  PROC DrawPart276()
    MoveL Offs(pOrigin,208.02,110.33,6.00),vTravel,z5,tPen\WObj:=wPaper;
    MoveL Offs(pOrigin,208.02,110.33,0.00),v60,z0,tPen\WObj:=wPaper;
    MoveL Offs(pOrigin,210.27,108.07,0.00),v40,fine,tPen\WObj:=wPaper;
    MoveL Offs(pOrigin,210.27,108.07,6.00),v60,z5,tPen\WObj:=wPaper;
    MoveL Offs(pOrigin,213.02,105.82,6.00),vTravel,z5,tPen\WObj:=wPaper;
    MoveL Offs(pOrigin,213.02,105.82,0.00),v60,z0,tPen\WObj:=wPaper;
    MoveL Offs(pOrigin,214.30,105.82,0.00),v40,fine,tPen\WObj:=wPaper;
    MoveL Offs(pOrigin,214.30,105.82,6.00),v60,z5,tPen\WObj:=wPaper;
    MoveL Offs(pOrigin,214.72,103.70,6.00),vTravel,z5,tPen\WObj:=wPaper;
    MoveL Offs(pOrigin,214.72,103.70,0.00),v60,z0,tPen\WObj:=wPaper;
    MoveL Offs(pOrigin,213.45,103.70,0.00),v40,z0,tPen\WObj:=wPaper;
    MoveL Offs(pOrigin,213.88,102.65,0.00),v40,z0,tPen\WObj:=wPaper;
    MoveL Offs(pOrigin,214.94,102.65,0.00),v40,fine,tPen\WObj:=wPaper;
    MoveL Offs(pOrigin,214.94,102.65,6.00),v60,z5,tPen\WObj:=wPaper;
    MoveL Offs(pOrigin,215.36,100.54,6.00),vTravel,z5,tPen\WObj:=wPaper;
    MoveL Offs(pOrigin,215.36,100.54,0.00),v60,z0,tPen\WObj:=wPaper;
    MoveL Offs(pOrigin,214.30,100.54,0.00),v40,z0,tPen\WObj:=wPaper;
    MoveL Offs(pOrigin,214.51,99.48,0.00),v40,z0,tPen\WObj:=wPaper;
    MoveL Offs(pOrigin,215.58,99.48,0.00),v40,z0,tPen\WObj:=wPaper;
    MoveL Offs(pOrigin,215.79,98.42,0.00),v40,z0,tPen\WObj:=wPaper;
    MoveL Offs(pOrigin,214.72,98.42,0.00),v40,fine,tPen\WObj:=wPaper;
    MoveL Offs(pOrigin,214.72,98.42,6.00),v60,z5,tPen\WObj:=wPaper;
    MoveL Offs(pOrigin,206.17,76.33,6.00),vTravel,z5,tPen\WObj:=wPaper;
    MoveL Offs(pOrigin,206.17,76.33,0.00),v60,z0,tPen\WObj:=wPaper;
    MoveL Offs(pOrigin,211.13,71.37,0.00),v40,z0,tPen\WObj:=wPaper;
    MoveL Offs(pOrigin,211.85,71.76,0.00),v40,z0,tPen\WObj:=wPaper;
    MoveL Offs(pOrigin,213.50,73.41,0.00),v40,fine,tPen\WObj:=wPaper;
    MoveL Offs(pOrigin,213.50,73.41,6.00),v60,z5,tPen\WObj:=wPaper;
    MoveL Offs(pOrigin,205.72,76.08,6.00),vTravel,z5,tPen\WObj:=wPaper;
    MoveL Offs(pOrigin,205.72,76.08,0.00),v60,z0,tPen\WObj:=wPaper;
    MoveL Offs(pOrigin,203.91,74.28,0.00),v40,fine,tPen\WObj:=wPaper;
    MoveL Offs(pOrigin,203.91,74.28,6.00),v60,z5,tPen\WObj:=wPaper;
    MoveL Offs(pOrigin,199.85,71.72,6.00),vTravel,z5,tPen\WObj:=wPaper;
    MoveL Offs(pOrigin,199.85,71.72,0.00),v60,z0,tPen\WObj:=wPaper;
    MoveL Offs(pOrigin,200.27,71.51,0.00),v40,z0,tPen\WObj:=wPaper;
    MoveL Offs(pOrigin,199.85,71.72,0.00),v40,fine,tPen\WObj:=wPaper;
    MoveL Offs(pOrigin,199.85,71.72,6.00),v60,z5,tPen\WObj:=wPaper;
    MoveL Offs(pOrigin,196.43,72.15,6.00),vTravel,z5,tPen\WObj:=wPaper;
    MoveL Offs(pOrigin,196.43,72.15,0.00),v60,z0,tPen\WObj:=wPaper;
    MoveL Offs(pOrigin,196.43,75.76,0.00),v40,fine,tPen\WObj:=wPaper;
    MoveL Offs(pOrigin,196.43,75.76,6.00),v60,z5,tPen\WObj:=wPaper;
    MoveL Offs(pOrigin,194.75,76.40,6.00),vTravel,z5,tPen\WObj:=wPaper;
    MoveL Offs(pOrigin,194.75,76.40,0.00),v60,z0,tPen\WObj:=wPaper;
    MoveL Offs(pOrigin,194.32,76.82,0.00),v40,z0,tPen\WObj:=wPaper;
    MoveL Offs(pOrigin,194.75,76.40,0.00),v40,z0,tPen\WObj:=wPaper;
    MoveL Offs(pOrigin,194.32,76.19,0.00),v40,z0,tPen\WObj:=wPaper;
    MoveL Offs(pOrigin,194.32,73.64,0.00),v40,z0,tPen\WObj:=wPaper;
    MoveL Offs(pOrigin,193.26,73.85,0.00),v40,z0,tPen\WObj:=wPaper;
    MoveL Offs(pOrigin,193.26,74.91,0.00),v40,fine,tPen\WObj:=wPaper;
    MoveL Offs(pOrigin,193.26,74.91,6.00),v60,z5,tPen\WObj:=wPaper;
    MoveL Offs(pOrigin,194.11,77.04,6.00),vTravel,z5,tPen\WObj:=wPaper;
    MoveL Offs(pOrigin,194.11,77.04,0.00),v60,z0,tPen\WObj:=wPaper;
    MoveL Offs(pOrigin,193.69,77.46,0.00),v40,z0,tPen\WObj:=wPaper;
    MoveL Offs(pOrigin,194.11,77.04,0.00),v40,z0,tPen\WObj:=wPaper;
    MoveL Offs(pOrigin,194.79,77.10,0.00),v40,z0,tPen\WObj:=wPaper;
    MoveL Offs(pOrigin,191.33,73.64,0.00),v40,fine,tPen\WObj:=wPaper;
    MoveL Offs(pOrigin,191.33,73.64,6.00),v60,z5,tPen\WObj:=wPaper;
    MoveL Offs(pOrigin,189.24,74.54,6.00),vTravel,z5,tPen\WObj:=wPaper;
    MoveL Offs(pOrigin,189.24,74.54,0.00),v60,z0,tPen\WObj:=wPaper;
    MoveL Offs(pOrigin,193.14,78.44,0.00),v40,z0,tPen\WObj:=wPaper;
    MoveL Offs(pOrigin,193.05,77.89,0.00),v40,z0,tPen\WObj:=wPaper;
    MoveL Offs(pOrigin,191.77,79.16,0.00),v40,z0,tPen\WObj:=wPaper;
    MoveL Offs(pOrigin,193.05,77.89,0.00),v40,z0,tPen\WObj:=wPaper;
    MoveL Offs(pOrigin,192.20,78.36,0.00),v40,z0,tPen\WObj:=wPaper;
    MoveL Offs(pOrigin,188.80,78.36,0.00),v40,fine,tPen\WObj:=wPaper;
    MoveL Offs(pOrigin,188.80,78.36,6.00),v60,z5,tPen\WObj:=wPaper;
    MoveL Offs(pOrigin,190.09,78.52,6.00),vTravel,z5,tPen\WObj:=wPaper;
    MoveL Offs(pOrigin,190.09,78.52,0.00),v60,z0,tPen\WObj:=wPaper;
    MoveL Offs(pOrigin,190.09,79.59,0.00),v40,z0,tPen\WObj:=wPaper;
    MoveL Offs(pOrigin,190.08,80.47,0.00),v40,z0,tPen\WObj:=wPaper;
    MoveL Offs(pOrigin,187.31,80.47,0.00),v40,z0,tPen\WObj:=wPaper;
    MoveL Offs(pOrigin,186.26,80.52,0.00),v40,z0,tPen\WObj:=wPaper;
    MoveL Offs(pOrigin,188.81,83.07,0.00),v40,z0,tPen\WObj:=wPaper;
    MoveL Offs(pOrigin,188.80,82.78,0.00),v40,z0,tPen\WObj:=wPaper;
    MoveL Offs(pOrigin,187.52,84.05,0.00),v40,z0,tPen\WObj:=wPaper;
    MoveL Offs(pOrigin,188.80,82.78,0.00),v40,z0,tPen\WObj:=wPaper;
    MoveL Offs(pOrigin,188.59,82.58,0.00),v40,z0,tPen\WObj:=wPaper;
    MoveL Offs(pOrigin,186.25,82.58,0.00),v40,fine,tPen\WObj:=wPaper;
    MoveL Offs(pOrigin,186.25,82.58,6.00),v60,z5,tPen\WObj:=wPaper;
    MoveL Offs(pOrigin,185.51,81.27,6.00),vTravel,z5,tPen\WObj:=wPaper;
    MoveL Offs(pOrigin,185.51,81.27,0.00),v60,z0,tPen\WObj:=wPaper;
    MoveL Offs(pOrigin,188.22,83.97,0.00),v40,fine,tPen\WObj:=wPaper;
    MoveL Offs(pOrigin,188.22,83.97,6.00),v60,z5,tPen\WObj:=wPaper;
    MoveL Offs(pOrigin,190.31,81.58,6.00),vTravel,z5,tPen\WObj:=wPaper;
    MoveL Offs(pOrigin,190.31,81.58,0.00),v60,z0,tPen\WObj:=wPaper;
    MoveL Offs(pOrigin,187.60,78.87,0.00),v40,fine,tPen\WObj:=wPaper;
    MoveL Offs(pOrigin,187.60,78.87,6.00),v60,z5,tPen\WObj:=wPaper;
    MoveL Offs(pOrigin,183.56,80.81,6.00),vTravel,z5,tPen\WObj:=wPaper;
    MoveL Offs(pOrigin,183.56,80.81,0.00),v60,z0,tPen\WObj:=wPaper;
    MoveL Offs(pOrigin,179.35,76.60,0.00),v40,z0,tPen\WObj:=wPaper;
    MoveL Offs(pOrigin,179.51,76.11,0.00),v40,z0,tPen\WObj:=wPaper;
    MoveL Offs(pOrigin,177.11,78.52,0.00),v40,z0,tPen\WObj:=wPaper;
    MoveL Offs(pOrigin,176.21,77.92,0.00),v40,z0,tPen\WObj:=wPaper;
    MoveL Offs(pOrigin,178.46,75.67,0.00),v40,fine,tPen\WObj:=wPaper;
    MoveL Offs(pOrigin,178.46,75.67,6.00),v60,z5,tPen\WObj:=wPaper;
    MoveL Offs(pOrigin,180.59,77.68,6.00),vTravel,z5,tPen\WObj:=wPaper;
    MoveL Offs(pOrigin,180.59,77.68,0.00),v60,z0,tPen\WObj:=wPaper;
    MoveL Offs(pOrigin,180.59,79.80,0.00),v40,fine,tPen\WObj:=wPaper;
    MoveL Offs(pOrigin,180.59,79.80,6.00),v60,z5,tPen\WObj:=wPaper;
    MoveL Offs(pOrigin,178.81,80.22,6.00),vTravel,z5,tPen\WObj:=wPaper;
    MoveL Offs(pOrigin,178.81,80.22,0.00),v60,z0,tPen\WObj:=wPaper;
    MoveL Offs(pOrigin,179.02,79.80,0.00),v40,z0,tPen\WObj:=wPaper;
    MoveL Offs(pOrigin,178.81,80.22,0.00),v40,fine,tPen\WObj:=wPaper;
    MoveL Offs(pOrigin,178.81,80.22,6.00),v60,z5,tPen\WObj:=wPaper;
    MoveL Offs(pOrigin,172.03,74.64,6.00),vTravel,z5,tPen\WObj:=wPaper;
    MoveL Offs(pOrigin,172.03,74.64,0.00),v60,z0,tPen\WObj:=wPaper;
    MoveL Offs(pOrigin,174.28,72.38,0.00),v40,fine,tPen\WObj:=wPaper;
    MoveL Offs(pOrigin,174.28,72.38,6.00),v60,z5,tPen\WObj:=wPaper;
    MoveL Offs(pOrigin,169.25,68.96,6.00),vTravel,z5,tPen\WObj:=wPaper;
    MoveL Offs(pOrigin,169.25,68.96,0.00),v60,z0,tPen\WObj:=wPaper;
    MoveL Offs(pOrigin,169.68,69.39,0.00),v40,z0,tPen\WObj:=wPaper;
    MoveL Offs(pOrigin,169.25,68.96,0.00),v40,fine,tPen\WObj:=wPaper;
    MoveL Offs(pOrigin,169.25,68.96,6.00),v60,z5,tPen\WObj:=wPaper;
    MoveL Offs(pOrigin,166.91,73.43,6.00),vTravel,z5,tPen\WObj:=wPaper;
    MoveL Offs(pOrigin,166.91,73.43,0.00),v60,z0,tPen\WObj:=wPaper;
    MoveL Offs(pOrigin,167.34,73.21,0.00),v40,z0,tPen\WObj:=wPaper;
    MoveL Offs(pOrigin,166.91,73.43,0.00),v40,fine,tPen\WObj:=wPaper;
    MoveL Offs(pOrigin,166.91,73.43,6.00),v60,z5,tPen\WObj:=wPaper;
    MoveL Offs(pOrigin,167.22,76.42,6.00),vTravel,z5,tPen\WObj:=wPaper;
    MoveL Offs(pOrigin,167.22,76.42,0.00),v60,z0,tPen\WObj:=wPaper;
  ENDPROC

  PROC DrawPart277()
    MoveL Offs(pOrigin,168.57,77.77,0.00),v40,z0,tPen\WObj:=wPaper;
    MoveL Offs(pOrigin,169.17,77.49,0.00),v40,z0,tPen\WObj:=wPaper;
    MoveL Offs(pOrigin,163.91,82.75,0.00),v40,z0,tPen\WObj:=wPaper;
    MoveL Offs(pOrigin,164.69,82.85,0.00),v40,z0,tPen\WObj:=wPaper;
    MoveL Offs(pOrigin,166.05,84.20,0.00),v40,fine,tPen\WObj:=wPaper;
    MoveL Offs(pOrigin,166.05,84.20,6.00),v60,z5,tPen\WObj:=wPaper;
    MoveL Offs(pOrigin,166.34,83.00,6.00),vTravel,z5,tPen\WObj:=wPaper;
    MoveL Offs(pOrigin,166.34,83.00,0.00),v60,z0,tPen\WObj:=wPaper;
    MoveL Offs(pOrigin,165.14,81.80,0.00),v40,fine,tPen\WObj:=wPaper;
    MoveL Offs(pOrigin,165.14,81.80,6.00),v60,z5,tPen\WObj:=wPaper;
    MoveL Offs(pOrigin,167.08,80.76,6.00),vTravel,z5,tPen\WObj:=wPaper;
    MoveL Offs(pOrigin,167.08,80.76,0.00),v60,z0,tPen\WObj:=wPaper;
    MoveL Offs(pOrigin,165.88,79.56,0.00),v40,fine,tPen\WObj:=wPaper;
    MoveL Offs(pOrigin,165.88,79.56,6.00),v60,z5,tPen\WObj:=wPaper;
    MoveL Offs(pOrigin,166.77,77.46,6.00),vTravel,z5,tPen\WObj:=wPaper;
    MoveL Offs(pOrigin,166.77,77.46,0.00),v60,z0,tPen\WObj:=wPaper;
    MoveL Offs(pOrigin,167.98,78.66,0.00),v40,fine,tPen\WObj:=wPaper;
    MoveL Offs(pOrigin,167.98,78.66,6.00),v60,z5,tPen\WObj:=wPaper;
    MoveL Offs(pOrigin,163.03,76.70,6.00),vTravel,z5,tPen\WObj:=wPaper;
    MoveL Offs(pOrigin,163.03,76.70,0.00),v60,z0,tPen\WObj:=wPaper;
    MoveL Offs(pOrigin,135.98,49.66,0.00),v40,z0,tPen\WObj:=wPaper;
    MoveL Offs(pOrigin,136.31,49.85,0.00),v40,z0,tPen\WObj:=wPaper;
    MoveL Offs(pOrigin,143.11,49.85,0.00),v40,fine,tPen\WObj:=wPaper;
    MoveL Offs(pOrigin,143.11,49.85,6.00),v60,z5,tPen\WObj:=wPaper;
    MoveL Offs(pOrigin,141.52,48.99,6.00),vTravel,z5,tPen\WObj:=wPaper;
    MoveL Offs(pOrigin,141.52,48.99,0.00),v60,z0,tPen\WObj:=wPaper;
    MoveL Offs(pOrigin,141.52,53.66,0.00),v40,z0,tPen\WObj:=wPaper;
    MoveL Offs(pOrigin,140.46,53.88,0.00),v40,z0,tPen\WObj:=wPaper;
    MoveL Offs(pOrigin,140.46,49.62,0.00),v40,z0,tPen\WObj:=wPaper;
    MoveL Offs(pOrigin,140.35,50.47,0.00),v40,z0,tPen\WObj:=wPaper;
    MoveL Offs(pOrigin,140.42,48.35,0.00),v40,z0,tPen\WObj:=wPaper;
    MoveL Offs(pOrigin,141.20,47.92,0.00),v40,fine,tPen\WObj:=wPaper;
    MoveL Offs(pOrigin,141.20,47.92,6.00),v60,z5,tPen\WObj:=wPaper;
    MoveL Offs(pOrigin,143.32,46.68,6.00),vTravel,z5,tPen\WObj:=wPaper;
    MoveL Offs(pOrigin,143.32,46.68,0.00),v60,z0,tPen\WObj:=wPaper;
    MoveL Offs(pOrigin,137.59,46.68,0.00),v40,z0,tPen\WObj:=wPaper;
    MoveL Offs(pOrigin,137.16,46.44,0.00),v40,z0,tPen\WObj:=wPaper;
    MoveL Offs(pOrigin,138.08,45.80,0.00),v40,z0,tPen\WObj:=wPaper;
    MoveL Offs(pOrigin,140.56,42.40,0.00),v40,z0,tPen\WObj:=wPaper;
    MoveL Offs(pOrigin,143.18,39.92,0.00),v40,z0,tPen\WObj:=wPaper;
    MoveL Offs(pOrigin,142.69,40.28,0.00),v40,z0,tPen\WObj:=wPaper;
    MoveL Offs(pOrigin,142.69,40.34,0.00),v40,z0,tPen\WObj:=wPaper;
    MoveL Offs(pOrigin,151.82,40.34,0.00),v40,z0,tPen\WObj:=wPaper;
    MoveL Offs(pOrigin,152.28,40.57,0.00),v40,z0,tPen\WObj:=wPaper;
    MoveL Offs(pOrigin,147.32,35.61,0.00),v40,z0,tPen\WObj:=wPaper;
    MoveL Offs(pOrigin,147.58,34.86,0.00),v40,z0,tPen\WObj:=wPaper;
    MoveL Offs(pOrigin,136.16,46.28,0.00),v40,z0,tPen\WObj:=wPaper;
    MoveL Offs(pOrigin,136.74,46.22,0.00),v40,z0,tPen\WObj:=wPaper;
    MoveL Offs(pOrigin,137.02,44.95,0.00),v40,z0,tPen\WObj:=wPaper;
    MoveL Offs(pOrigin,138.37,42.40,0.00),v40,z0,tPen\WObj:=wPaper;
    MoveL Offs(pOrigin,140.21,39.85,0.00),v40,z0,tPen\WObj:=wPaper;
    MoveL Offs(pOrigin,141.84,38.36,0.00),v40,z0,tPen\WObj:=wPaper;
    MoveL Offs(pOrigin,141.84,38.36,0.00),v40,z0,tPen\WObj:=wPaper;
    MoveL Offs(pOrigin,146.09,37.09,0.00),v40,z0,tPen\WObj:=wPaper;
    MoveL Offs(pOrigin,150.98,37.30,0.00),v40,z0,tPen\WObj:=wPaper;
    MoveL Offs(pOrigin,152.89,37.80,0.00),v40,z0,tPen\WObj:=wPaper;
    MoveL Offs(pOrigin,153.10,38.15,0.00),v40,z0,tPen\WObj:=wPaper;
    MoveL Offs(pOrigin,152.89,38.58,0.00),v40,z0,tPen\WObj:=wPaper;
    MoveL Offs(pOrigin,148.00,38.15,0.00),v40,z0,tPen\WObj:=wPaper;
    MoveL Offs(pOrigin,144.39,39.14,0.00),v40,z0,tPen\WObj:=wPaper;
    MoveL Offs(pOrigin,143.75,39.64,0.00),v40,z0,tPen\WObj:=wPaper;
    MoveL Offs(pOrigin,144.18,39.42,0.00),v40,z0,tPen\WObj:=wPaper;
    MoveL Offs(pOrigin,144.60,39.21,0.00),v40,z0,tPen\WObj:=wPaper;
    MoveL Offs(pOrigin,144.18,39.42,0.00),v40,z0,tPen\WObj:=wPaper;
    MoveL Offs(pOrigin,143.63,40.49,0.00),v40,z0,tPen\WObj:=wPaper;
    MoveL Offs(pOrigin,143.63,44.74,0.00),v40,fine,tPen\WObj:=wPaper;
    MoveL Offs(pOrigin,143.63,44.74,6.00),v60,z5,tPen\WObj:=wPaper;
    MoveL Offs(pOrigin,145.25,43.99,6.00),vTravel,z5,tPen\WObj:=wPaper;
    MoveL Offs(pOrigin,145.25,43.99,0.00),v60,z0,tPen\WObj:=wPaper;
    MoveL Offs(pOrigin,141.79,40.54,0.00),v40,z0,tPen\WObj:=wPaper;
    MoveL Offs(pOrigin,142.05,40.70,0.00),v40,z0,tPen\WObj:=wPaper;
    MoveL Offs(pOrigin,141.62,41.12,0.00),v40,z0,tPen\WObj:=wPaper;
    MoveL Offs(pOrigin,142.05,40.70,0.00),v40,z0,tPen\WObj:=wPaper;
    MoveL Offs(pOrigin,142.57,41.12,0.00),v40,z0,tPen\WObj:=wPaper;
    MoveL Offs(pOrigin,142.57,42.40,0.00),v40,z0,tPen\WObj:=wPaper;
    MoveL Offs(pOrigin,141.52,42.19,0.00),v40,z0,tPen\WObj:=wPaper;
    MoveL Offs(pOrigin,141.52,43.25,0.00),v40,fine,tPen\WObj:=wPaper;
    MoveL Offs(pOrigin,141.52,43.25,6.00),v60,z5,tPen\WObj:=wPaper;
    MoveL Offs(pOrigin,141.04,39.78,6.00),vTravel,z5,tPen\WObj:=wPaper;
    MoveL Offs(pOrigin,141.04,39.78,0.00),v60,z0,tPen\WObj:=wPaper;
    MoveL Offs(pOrigin,140.29,39.03,0.00),v40,z0,tPen\WObj:=wPaper;
    MoveL Offs(pOrigin,140.56,39.42,0.00),v40,z0,tPen\WObj:=wPaper;
    MoveL Offs(pOrigin,140.35,39.85,0.00),v40,z0,tPen\WObj:=wPaper;
    MoveL Offs(pOrigin,140.56,39.42,0.00),v40,fine,tPen\WObj:=wPaper;
    MoveL Offs(pOrigin,140.56,39.42,6.00),v60,z5,tPen\WObj:=wPaper;
    MoveL Offs(pOrigin,141.79,39.04,6.00),vTravel,z5,tPen\WObj:=wPaper;
    MoveL Offs(pOrigin,141.79,39.04,0.00),v60,z0,tPen\WObj:=wPaper;
    MoveL Offs(pOrigin,138.93,36.18,0.00),v40,z0,tPen\WObj:=wPaper;
    MoveL Offs(pOrigin,139.49,35.49,0.00),v40,z0,tPen\WObj:=wPaper;
    MoveL Offs(pOrigin,135.43,39.55,0.00),v40,z0,tPen\WObj:=wPaper;
    MoveL Offs(pOrigin,135.65,38.87,0.00),v40,z0,tPen\WObj:=wPaper;
    MoveL Offs(pOrigin,133.69,36.92,0.00),v40,z0,tPen\WObj:=wPaper;
    MoveL Offs(pOrigin,134.13,37.51,0.00),v40,z0,tPen\WObj:=wPaper;
    MoveL Offs(pOrigin,134.13,38.79,0.00),v40,z0,tPen\WObj:=wPaper;
    MoveL Offs(pOrigin,133.76,39.29,0.00),v40,z0,tPen\WObj:=wPaper;
    MoveL Offs(pOrigin,103.16,39.29,0.00),v40,z0,tPen\WObj:=wPaper;
    MoveL Offs(pOrigin,103.14,39.22,0.00),v40,z0,tPen\WObj:=wPaper;
    MoveL Offs(pOrigin,104.64,40.72,0.00),v40,z0,tPen\WObj:=wPaper;
    MoveL Offs(pOrigin,104.22,40.34,0.00),v40,z0,tPen\WObj:=wPaper;
    MoveL Offs(pOrigin,99.98,40.34,0.00),v40,z0,tPen\WObj:=wPaper;
    MoveL Offs(pOrigin,99.70,40.26,0.00),v40,z0,tPen\WObj:=wPaper;
    MoveL Offs(pOrigin,101.20,41.76,0.00),v40,z0,tPen\WObj:=wPaper;
    MoveL Offs(pOrigin,101.72,41.90,0.00),v40,z0,tPen\WObj:=wPaper;
    MoveL Offs(pOrigin,109.23,34.38,0.00),v40,fine,tPen\WObj:=wPaper;
    MoveL Offs(pOrigin,109.23,34.38,6.00),v60,z5,tPen\WObj:=wPaper;
    MoveL Offs(pOrigin,107.89,34.24,6.00),vTravel,z5,tPen\WObj:=wPaper;
    MoveL Offs(pOrigin,107.89,34.24,0.00),v60,z0,tPen\WObj:=wPaper;
    MoveL Offs(pOrigin,98.72,43.40,0.00),v40,z0,tPen\WObj:=wPaper;
    MoveL Offs(pOrigin,99.11,42.65,0.00),v40,z0,tPen\WObj:=wPaper;
    MoveL Offs(pOrigin,97.76,41.30,0.00),v40,z0,tPen\WObj:=wPaper;
    MoveL Offs(pOrigin,97.85,41.40,0.00),v40,z0,tPen\WObj:=wPaper;
    MoveL Offs(pOrigin,100.61,41.40,0.00),v40,z0,tPen\WObj:=wPaper;
    MoveL Offs(pOrigin,100.16,42.21,0.00),v40,z0,tPen\WObj:=wPaper;
    MoveL Offs(pOrigin,98.65,40.70,0.00),v40,z0,tPen\WObj:=wPaper;
    MoveL Offs(pOrigin,99.34,40.70,0.00),v40,z0,tPen\WObj:=wPaper;
    MoveL Offs(pOrigin,99.76,40.49,0.00),v40,z0,tPen\WObj:=wPaper;
    MoveL Offs(pOrigin,99.34,40.70,0.00),v40,fine,tPen\WObj:=wPaper;
    MoveL Offs(pOrigin,99.34,40.70,6.00),v60,z5,tPen\WObj:=wPaper;
    MoveL Offs(pOrigin,99.63,39.51,6.00),vTravel,z5,tPen\WObj:=wPaper;
    MoveL Offs(pOrigin,99.63,39.51,0.00),v60,z0,tPen\WObj:=wPaper;
  ENDPROC

  PROC DrawPart278()
    MoveL Offs(pOrigin,91.97,47.17,0.00),v40,z0,tPen\WObj:=wPaper;
    MoveL Offs(pOrigin,92.83,46.83,0.00),v40,z0,tPen\WObj:=wPaper;
    MoveL Offs(pOrigin,94.48,48.48,0.00),v40,z0,tPen\WObj:=wPaper;
    MoveL Offs(pOrigin,94.24,48.79,0.00),v40,z0,tPen\WObj:=wPaper;
    MoveL Offs(pOrigin,92.54,48.79,0.00),v40,z0,tPen\WObj:=wPaper;
    MoveL Offs(pOrigin,92.94,48.78,0.00),v40,z0,tPen\WObj:=wPaper;
    MoveL Offs(pOrigin,92.94,57.06,0.00),v40,z0,tPen\WObj:=wPaper;
    MoveL Offs(pOrigin,93.18,57.28,0.00),v40,z0,tPen\WObj:=wPaper;
    MoveL Offs(pOrigin,92.61,57.49,0.00),v40,z0,tPen\WObj:=wPaper;
    MoveL Offs(pOrigin,91.90,59.61,0.00),v40,z0,tPen\WObj:=wPaper;
    MoveL Offs(pOrigin,90.62,66.62,0.00),v40,z0,tPen\WObj:=wPaper;
    MoveL Offs(pOrigin,90.84,70.03,0.00),v40,z0,tPen\WObj:=wPaper;
    MoveL Offs(pOrigin,92.25,74.49,0.00),v40,z0,tPen\WObj:=wPaper;
    MoveL Offs(pOrigin,96.22,81.07,0.00),v40,z0,tPen\WObj:=wPaper;
    MoveL Offs(pOrigin,98.63,87.03,0.00),v40,z0,tPen\WObj:=wPaper;
    MoveL Offs(pOrigin,99.97,89.36,0.00),v40,z0,tPen\WObj:=wPaper;
    MoveL Offs(pOrigin,102.95,92.34,0.00),v40,z0,tPen\WObj:=wPaper;
    MoveL Offs(pOrigin,111.17,97.72,0.00),v40,z0,tPen\WObj:=wPaper;
    MoveL Offs(pOrigin,111.45,98.71,0.00),v40,z0,tPen\WObj:=wPaper;
    MoveL Offs(pOrigin,111.45,98.71,0.00),v40,z0,tPen\WObj:=wPaper;
    MoveL Offs(pOrigin,119.74,103.25,0.00),v40,z0,tPen\WObj:=wPaper;
    MoveL Offs(pOrigin,120.80,103.39,0.00),v40,fine,tPen\WObj:=wPaper;
    MoveL Offs(pOrigin,120.80,103.39,6.00),v60,z5,tPen\WObj:=wPaper;
    MoveL Offs(pOrigin,119.06,102.21,6.00),vTravel,z5,tPen\WObj:=wPaper;
    MoveL Offs(pOrigin,119.06,102.21,0.00),v60,z0,tPen\WObj:=wPaper;
    MoveL Offs(pOrigin,118.16,103.11,0.00),v40,z0,tPen\WObj:=wPaper;
    MoveL Offs(pOrigin,117.11,102.67,0.00),v40,z0,tPen\WObj:=wPaper;
    MoveL Offs(pOrigin,118.16,101.62,0.00),v40,z0,tPen\WObj:=wPaper;
    MoveL Offs(pOrigin,117.27,101.02,0.00),v40,z0,tPen\WObj:=wPaper;
    MoveL Offs(pOrigin,116.07,102.22,0.00),v40,z0,tPen\WObj:=wPaper;
    MoveL Offs(pOrigin,115.17,101.62,0.00),v40,z0,tPen\WObj:=wPaper;
    MoveL Offs(pOrigin,116.52,100.27,0.00),v40,z0,tPen\WObj:=wPaper;
    MoveL Offs(pOrigin,115.62,99.68,0.00),v40,z0,tPen\WObj:=wPaper;
    MoveL Offs(pOrigin,114.12,101.18,0.00),v40,z0,tPen\WObj:=wPaper;
    MoveL Offs(pOrigin,113.67,100.52,0.00),v40,z0,tPen\WObj:=wPaper;
    MoveL Offs(pOrigin,109.31,96.16,0.00),v40,z0,tPen\WObj:=wPaper;
    MoveL Offs(pOrigin,109.35,95.50,0.00),v40,z0,tPen\WObj:=wPaper;
    MoveL Offs(pOrigin,103.94,100.91,0.00),v40,z0,tPen\WObj:=wPaper;
    MoveL Offs(pOrigin,104.86,100.54,0.00),v40,z0,tPen\WObj:=wPaper;
    MoveL Offs(pOrigin,106.35,100.54,0.00),v40,z0,tPen\WObj:=wPaper;
    MoveL Offs(pOrigin,106.62,99.45,0.00),v40,z0,tPen\WObj:=wPaper;
    MoveL Offs(pOrigin,102.72,95.54,0.00),v40,z0,tPen\WObj:=wPaper;
    MoveL Offs(pOrigin,102.16,95.22,0.00),v40,z0,tPen\WObj:=wPaper;
    MoveL Offs(pOrigin,104.86,92.52,0.00),v40,z0,tPen\WObj:=wPaper;
    MoveL Offs(pOrigin,104.81,93.15,0.00),v40,z0,tPen\WObj:=wPaper;
    MoveL Offs(pOrigin,110.67,99.01,0.00),v40,z0,tPen\WObj:=wPaper;
    MoveL Offs(pOrigin,110.23,99.09,0.00),v40,z0,tPen\WObj:=wPaper;
    MoveL Offs(pOrigin,111.89,97.44,0.00),v40,z0,tPen\WObj:=wPaper;
    MoveL Offs(pOrigin,111.14,96.69,0.00),v40,z0,tPen\WObj:=wPaper;
    MoveL Offs(pOrigin,109.34,98.50,0.00),v40,z0,tPen\WObj:=wPaper;
    MoveL Offs(pOrigin,109.32,97.86,0.00),v40,z0,tPen\WObj:=wPaper;
    MoveL Offs(pOrigin,109.75,98.07,0.00),v40,z0,tPen\WObj:=wPaper;
    MoveL Offs(pOrigin,109.32,97.86,0.00),v40,z0,tPen\WObj:=wPaper;
    MoveL Offs(pOrigin,109.54,96.80,0.00),v40,z0,tPen\WObj:=wPaper;
    MoveL Offs(pOrigin,109.96,97.01,0.00),v40,z0,tPen\WObj:=wPaper;
    MoveL Offs(pOrigin,109.54,96.80,0.00),v40,z0,tPen\WObj:=wPaper;
    MoveL Offs(pOrigin,110.24,96.10,0.00),v40,z0,tPen\WObj:=wPaper;
    MoveL Offs(pOrigin,104.38,101.96,0.00),v40,fine,tPen\WObj:=wPaper;
    MoveL Offs(pOrigin,104.38,101.96,6.00),v60,z5,tPen\WObj:=wPaper;
    MoveL Offs(pOrigin,105.50,102.65,6.00),vTravel,z5,tPen\WObj:=wPaper;
    MoveL Offs(pOrigin,105.50,102.65,0.00),v60,z0,tPen\WObj:=wPaper;
    MoveL Offs(pOrigin,106.99,102.65,0.00),v40,z0,tPen\WObj:=wPaper;
    MoveL Offs(pOrigin,107.20,103.70,0.00),v40,z0,tPen\WObj:=wPaper;
    MoveL Offs(pOrigin,105.93,103.70,0.00),v40,z0,tPen\WObj:=wPaper;
    MoveL Offs(pOrigin,105.44,104.24,0.00),v40,z0,tPen\WObj:=wPaper;
    MoveL Offs(pOrigin,110.25,109.05,0.00),v40,z0,tPen\WObj:=wPaper;
    MoveL Offs(pOrigin,109.75,108.98,0.00),v40,z0,tPen\WObj:=wPaper;
    MoveL Offs(pOrigin,108.26,108.98,0.00),v40,z0,tPen\WObj:=wPaper;
    MoveL Offs(pOrigin,107.62,108.70,0.00),v40,z0,tPen\WObj:=wPaper;
    MoveL Offs(pOrigin,108.05,109.34,0.00),v40,z0,tPen\WObj:=wPaper;
    MoveL Offs(pOrigin,107.62,108.70,0.00),v40,z0,tPen\WObj:=wPaper;
    MoveL Offs(pOrigin,107.62,107.93,0.00),v40,z0,tPen\WObj:=wPaper;
    MoveL Offs(pOrigin,109.11,107.93,0.00),v40,z0,tPen\WObj:=wPaper;
    MoveL Offs(pOrigin,108.90,107.21,0.00),v40,z0,tPen\WObj:=wPaper;
    MoveL Offs(pOrigin,109.11,107.64,0.00),v40,z0,tPen\WObj:=wPaper;
    MoveL Offs(pOrigin,108.90,107.21,0.00),v40,z0,tPen\WObj:=wPaper;
    MoveL Offs(pOrigin,108.48,106.87,0.00),v40,z0,tPen\WObj:=wPaper;
    MoveL Offs(pOrigin,107.20,106.87,0.00),v40,z0,tPen\WObj:=wPaper;
    MoveL Offs(pOrigin,106.31,107.49,0.00),v40,z0,tPen\WObj:=wPaper;
    MoveL Offs(pOrigin,110.52,103.29,0.00),v40,z0,tPen\WObj:=wPaper;
    MoveL Offs(pOrigin,111.27,104.03,0.00),v40,z0,tPen\WObj:=wPaper;
    MoveL Offs(pOrigin,106.76,108.54,0.00),v40,z0,tPen\WObj:=wPaper;
    MoveL Offs(pOrigin,107.35,109.44,0.00),v40,z0,tPen\WObj:=wPaper;
    MoveL Offs(pOrigin,111.86,104.93,0.00),v40,z0,tPen\WObj:=wPaper;
    MoveL Offs(pOrigin,112.46,105.83,0.00),v40,z0,tPen\WObj:=wPaper;
    MoveL Offs(pOrigin,107.95,110.34,0.00),v40,z0,tPen\WObj:=wPaper;
    MoveL Offs(pOrigin,107.85,109.64,0.00),v40,z0,tPen\WObj:=wPaper;
    MoveL Offs(pOrigin,117.62,119.41,0.00),v40,z0,tPen\WObj:=wPaper;
    MoveL Offs(pOrigin,117.19,119.54,0.00),v40,z0,tPen\WObj:=wPaper;
    MoveL Offs(pOrigin,115.91,119.54,0.00),v40,fine,tPen\WObj:=wPaper;
    MoveL Offs(pOrigin,115.91,119.54,6.00),v60,z5,tPen\WObj:=wPaper;
    MoveL Offs(pOrigin,116.98,123.77,6.00),vTravel,z5,tPen\WObj:=wPaper;
    MoveL Offs(pOrigin,116.98,123.77,0.00),v60,z0,tPen\WObj:=wPaper;
    MoveL Offs(pOrigin,118.04,123.77,0.00),v40,fine,tPen\WObj:=wPaper;
    MoveL Offs(pOrigin,118.04,123.77,6.00),v60,z5,tPen\WObj:=wPaper;
    MoveL Offs(pOrigin,119.14,124.53,6.00),vTravel,z5,tPen\WObj:=wPaper;
    MoveL Offs(pOrigin,119.14,124.53,0.00),v60,z0,tPen\WObj:=wPaper;
    MoveL Offs(pOrigin,116.44,127.24,0.00),v40,fine,tPen\WObj:=wPaper;
    MoveL Offs(pOrigin,116.44,127.24,6.00),v60,z5,tPen\WObj:=wPaper;
    MoveL Offs(pOrigin,116.58,128.58,6.00),vTravel,z5,tPen\WObj:=wPaper;
    MoveL Offs(pOrigin,116.58,128.58,0.00),v60,z0,tPen\WObj:=wPaper;
    MoveL Offs(pOrigin,119.44,125.73,0.00),v40,z0,tPen\WObj:=wPaper;
    MoveL Offs(pOrigin,118.46,125.88,0.00),v40,z0,tPen\WObj:=wPaper;
    MoveL Offs(pOrigin,117.40,125.88,0.00),v40,fine,tPen\WObj:=wPaper;
    MoveL Offs(pOrigin,117.40,125.88,6.00),v60,z5,tPen\WObj:=wPaper;
    MoveL Offs(pOrigin,117.61,127.99,6.00),vTravel,z5,tPen\WObj:=wPaper;
    MoveL Offs(pOrigin,117.61,127.99,0.00),v60,z0,tPen\WObj:=wPaper;
    MoveL Offs(pOrigin,118.89,127.99,0.00),v40,z0,tPen\WObj:=wPaper;
    MoveL Offs(pOrigin,119.88,128.27,0.00),v40,z0,tPen\WObj:=wPaper;
    MoveL Offs(pOrigin,117.48,130.68,0.00),v40,z0,tPen\WObj:=wPaper;
    MoveL Offs(pOrigin,118.04,130.59,0.00),v40,z0,tPen\WObj:=wPaper;
    MoveL Offs(pOrigin,118.25,131.01,0.00),v40,z0,tPen\WObj:=wPaper;
    MoveL Offs(pOrigin,118.04,130.59,0.00),v40,z0,tPen\WObj:=wPaper;
    MoveL Offs(pOrigin,118.25,130.10,0.00),v40,z0,tPen\WObj:=wPaper;
    MoveL Offs(pOrigin,119.52,130.10,0.00),v40,z0,tPen\WObj:=wPaper;
    MoveL Offs(pOrigin,120.33,129.32,0.00),v40,z0,tPen\WObj:=wPaper;
    MoveL Offs(pOrigin,117.92,131.73,0.00),v40,fine,tPen\WObj:=wPaper;
    MoveL Offs(pOrigin,117.92,131.73,6.00),v60,z5,tPen\WObj:=wPaper;
    MoveL Offs(pOrigin,117.03,129.63,6.00),vTravel,z5,tPen\WObj:=wPaper;
    MoveL Offs(pOrigin,117.03,129.63,0.00),v60,z0,tPen\WObj:=wPaper;
  ENDPROC

  PROC DrawPart279()
    MoveL Offs(pOrigin,119.58,127.08,0.00),v40,fine,tPen\WObj:=wPaper;
    MoveL Offs(pOrigin,119.58,127.08,6.00),v60,z5,tPen\WObj:=wPaper;
    MoveL Offs(pOrigin,112.58,116.16,6.00),vTravel,z5,tPen\WObj:=wPaper;
    MoveL Offs(pOrigin,112.58,116.16,0.00),v60,z0,tPen\WObj:=wPaper;
    MoveL Offs(pOrigin,114.83,113.91,0.00),v40,z0,tPen\WObj:=wPaper;
    MoveL Offs(pOrigin,114.21,114.44,0.00),v40,z0,tPen\WObj:=wPaper;
    MoveL Offs(pOrigin,115.06,115.29,0.00),v40,z0,tPen\WObj:=wPaper;
    MoveL Offs(pOrigin,114.21,114.44,0.00),v40,z0,tPen\WObj:=wPaper;
    MoveL Offs(pOrigin,114.00,114.26,0.00),v40,z0,tPen\WObj:=wPaper;
    MoveL Offs(pOrigin,112.30,114.26,0.00),v40,z0,tPen\WObj:=wPaper;
    MoveL Offs(pOrigin,111.98,115.27,0.00),v40,z0,tPen\WObj:=wPaper;
    MoveL Offs(pOrigin,114.23,113.01,0.00),v40,z0,tPen\WObj:=wPaper;
    MoveL Offs(pOrigin,113.34,112.42,0.00),v40,z0,tPen\WObj:=wPaper;
    MoveL Offs(pOrigin,111.08,114.67,0.00),v40,z0,tPen\WObj:=wPaper;
    MoveL Offs(pOrigin,110.49,113.77,0.00),v40,z0,tPen\WObj:=wPaper;
    MoveL Offs(pOrigin,112.74,111.52,0.00),v40,z0,tPen\WObj:=wPaper;
    MoveL Offs(pOrigin,112.09,112.15,0.00),v40,z0,tPen\WObj:=wPaper;
    MoveL Offs(pOrigin,110.39,112.15,0.00),v40,z0,tPen\WObj:=wPaper;
    MoveL Offs(pOrigin,110.18,112.31,0.00),v40,z0,tPen\WObj:=wPaper;
    MoveL Offs(pOrigin,110.39,112.74,0.00),v40,z0,tPen\WObj:=wPaper;
    MoveL Offs(pOrigin,110.18,112.31,0.00),v40,z0,tPen\WObj:=wPaper;
    MoveL Offs(pOrigin,109.89,112.88,0.00),v40,z0,tPen\WObj:=wPaper;
    MoveL Offs(pOrigin,111.99,110.77,0.00),v40,z0,tPen\WObj:=wPaper;
    MoveL Offs(pOrigin,111.45,111.25,0.00),v40,z0,tPen\WObj:=wPaper;
    MoveL Offs(pOrigin,112.09,111.89,0.00),v40,z0,tPen\WObj:=wPaper;
    MoveL Offs(pOrigin,111.45,111.25,0.00),v40,z0,tPen\WObj:=wPaper;
    MoveL Offs(pOrigin,111.24,111.10,0.00),v40,z0,tPen\WObj:=wPaper;
    MoveL Offs(pOrigin,109.75,111.10,0.00),v40,z0,tPen\WObj:=wPaper;
    MoveL Offs(pOrigin,109.32,111.25,0.00),v40,z0,tPen\WObj:=wPaper;
    MoveL Offs(pOrigin,109.54,111.68,0.00),v40,z0,tPen\WObj:=wPaper;
    MoveL Offs(pOrigin,109.32,111.25,0.00),v40,z0,tPen\WObj:=wPaper;
    MoveL Offs(pOrigin,108.55,111.23,0.00),v40,z0,tPen\WObj:=wPaper;
    MoveL Offs(pOrigin,110.80,108.98,0.00),v40,z0,tPen\WObj:=wPaper;
    MoveL Offs(pOrigin,111.55,108.23,0.00),v40,z0,tPen\WObj:=wPaper;
    MoveL Offs(pOrigin,113.36,106.42,0.00),v40,z0,tPen\WObj:=wPaper;
    MoveL Offs(pOrigin,113.95,107.32,0.00),v40,z0,tPen\WObj:=wPaper;
    MoveL Offs(pOrigin,112.15,109.12,0.00),v40,z0,tPen\WObj:=wPaper;
    MoveL Offs(pOrigin,111.40,109.88,0.00),v40,z0,tPen\WObj:=wPaper;
    MoveL Offs(pOrigin,109.14,112.13,0.00),v40,fine,tPen\WObj:=wPaper;
    MoveL Offs(pOrigin,109.14,112.13,6.00),v60,z5,tPen\WObj:=wPaper;
    MoveL Offs(pOrigin,110.60,112.95,6.00),vTravel,z5,tPen\WObj:=wPaper;
    MoveL Offs(pOrigin,110.60,112.95,0.00),v60,z0,tPen\WObj:=wPaper;
    MoveL Offs(pOrigin,112.09,114.44,0.00),v40,z0,tPen\WObj:=wPaper;
    MoveL Offs(pOrigin,110.60,112.95,0.00),v40,z0,tPen\WObj:=wPaper;
    MoveL Offs(pOrigin,111.45,113.21,0.00),v40,z0,tPen\WObj:=wPaper;
    MoveL Offs(pOrigin,112.94,113.21,0.00),v40,z0,tPen\WObj:=wPaper;
    MoveL Offs(pOrigin,112.72,112.74,0.00),v40,z0,tPen\WObj:=wPaper;
    MoveL Offs(pOrigin,113.57,113.59,0.00),v40,z0,tPen\WObj:=wPaper;
    MoveL Offs(pOrigin,112.72,112.74,0.00),v40,fine,tPen\WObj:=wPaper;
    MoveL Offs(pOrigin,112.72,112.74,6.00),v60,z5,tPen\WObj:=wPaper;
    MoveL Offs(pOrigin,114.69,111.06,6.00),vTravel,z5,tPen\WObj:=wPaper;
    MoveL Offs(pOrigin,114.69,111.06,0.00),v60,z0,tPen\WObj:=wPaper;
    MoveL Offs(pOrigin,116.49,109.26,0.00),v40,z0,tPen\WObj:=wPaper;
    MoveL Offs(pOrigin,117.39,109.86,0.00),v40,z0,tPen\WObj:=wPaper;
    MoveL Offs(pOrigin,115.59,111.66,0.00),v40,z0,tPen\WObj:=wPaper;
    MoveL Offs(pOrigin,116.63,112.11,0.00),v40,z0,tPen\WObj:=wPaper;
    MoveL Offs(pOrigin,118.44,110.30,0.00),v40,z0,tPen\WObj:=wPaper;
    MoveL Offs(pOrigin,119.48,110.75,0.00),v40,z0,tPen\WObj:=wPaper;
    MoveL Offs(pOrigin,117.53,112.70,0.00),v40,z0,tPen\WObj:=wPaper;
    MoveL Offs(pOrigin,117.90,112.22,0.00),v40,z0,tPen\WObj:=wPaper;
    MoveL Offs(pOrigin,108.58,102.90,0.00),v40,z0,tPen\WObj:=wPaper;
    MoveL Offs(pOrigin,108.13,103.95,0.00),v40,z0,tPen\WObj:=wPaper;
    MoveL Offs(pOrigin,103.93,99.74,0.00),v40,z0,tPen\WObj:=wPaper;
    MoveL Offs(pOrigin,103.49,99.86,0.00),v40,z0,tPen\WObj:=wPaper;
    MoveL Offs(pOrigin,108.45,94.90,0.00),v40,fine,tPen\WObj:=wPaper;
    MoveL Offs(pOrigin,108.45,94.90,6.00),v60,z5,tPen\WObj:=wPaper;
    MoveL Offs(pOrigin,108.48,96.31,6.00),vTravel,z5,tPen\WObj:=wPaper;
    MoveL Offs(pOrigin,108.48,96.31,0.00),v60,z0,tPen\WObj:=wPaper;
    MoveL Offs(pOrigin,107.41,96.31,0.00),v40,z0,tPen\WObj:=wPaper;
    MoveL Offs(pOrigin,107.41,96.80,0.00),v40,z0,tPen\WObj:=wPaper;
    MoveL Offs(pOrigin,107.84,97.01,0.00),v40,z0,tPen\WObj:=wPaper;
    MoveL Offs(pOrigin,107.41,96.80,0.00),v40,z0,tPen\WObj:=wPaper;
    MoveL Offs(pOrigin,107.51,97.35,0.00),v40,z0,tPen\WObj:=wPaper;
    MoveL Offs(pOrigin,95.79,85.63,0.00),v40,z0,tPen\WObj:=wPaper;
    MoveL Offs(pOrigin,95.44,85.51,0.00),v40,z0,tPen\WObj:=wPaper;
    MoveL Offs(pOrigin,98.00,82.95,0.00),v40,z0,tPen\WObj:=wPaper;
    MoveL Offs(pOrigin,97.43,83.64,0.00),v40,z0,tPen\WObj:=wPaper;
    MoveL Offs(pOrigin,95.72,83.64,0.00),v40,z0,tPen\WObj:=wPaper;
    MoveL Offs(pOrigin,95.00,84.46,0.00),v40,z0,tPen\WObj:=wPaper;
    MoveL Offs(pOrigin,102.21,77.25,0.00),v40,z0,tPen\WObj:=wPaper;
    MoveL Offs(pOrigin,101.61,76.35,0.00),v40,z0,tPen\WObj:=wPaper;
    MoveL Offs(pOrigin,94.55,83.41,0.00),v40,z0,tPen\WObj:=wPaper;
    MoveL Offs(pOrigin,94.11,82.37,0.00),v40,z0,tPen\WObj:=wPaper;
    MoveL Offs(pOrigin,100.72,75.75,0.00),v40,z0,tPen\WObj:=wPaper;
    MoveL Offs(pOrigin,99.76,75.97,0.00),v40,z0,tPen\WObj:=wPaper;
    MoveL Offs(pOrigin,100.61,76.82,0.00),v40,z0,tPen\WObj:=wPaper;
    MoveL Offs(pOrigin,99.76,75.97,0.00),v40,z0,tPen\WObj:=wPaper;
    MoveL Offs(pOrigin,99.97,75.01,0.00),v40,z0,tPen\WObj:=wPaper;
    MoveL Offs(pOrigin,93.51,81.47,0.00),v40,z0,tPen\WObj:=wPaper;
    MoveL Offs(pOrigin,94.45,81.50,0.00),v40,z0,tPen\WObj:=wPaper;
    MoveL Offs(pOrigin,94.66,81.93,0.00),v40,z0,tPen\WObj:=wPaper;
    MoveL Offs(pOrigin,94.45,81.50,0.00),v40,z0,tPen\WObj:=wPaper;
    MoveL Offs(pOrigin,94.66,81.53,0.00),v40,z0,tPen\WObj:=wPaper;
    MoveL Offs(pOrigin,96.36,81.53,0.00),v40,z0,tPen\WObj:=wPaper;
    MoveL Offs(pOrigin,96.57,82.14,0.00),v40,z0,tPen\WObj:=wPaper;
    MoveL Offs(pOrigin,96.79,82.56,0.00),v40,z0,tPen\WObj:=wPaper;
    MoveL Offs(pOrigin,96.57,82.14,0.00),v40,fine,tPen\WObj:=wPaper;
    MoveL Offs(pOrigin,96.57,82.14,6.00),v60,z5,tPen\WObj:=wPaper;
    MoveL Offs(pOrigin,95.72,80.47,6.00),vTravel,z5,tPen\WObj:=wPaper;
    MoveL Offs(pOrigin,95.72,80.47,0.00),v60,z0,tPen\WObj:=wPaper;
    MoveL Offs(pOrigin,94.24,80.47,0.00),v40,z0,tPen\WObj:=wPaper;
    MoveL Offs(pOrigin,93.60,80.01,0.00),v40,z0,tPen\WObj:=wPaper;
    MoveL Offs(pOrigin,93.81,80.44,0.00),v40,z0,tPen\WObj:=wPaper;
    MoveL Offs(pOrigin,93.60,80.01,0.00),v40,z0,tPen\WObj:=wPaper;
    MoveL Offs(pOrigin,93.39,79.42,0.00),v40,z0,tPen\WObj:=wPaper;
    MoveL Offs(pOrigin,95.09,79.42,0.00),v40,z0,tPen\WObj:=wPaper;
    MoveL Offs(pOrigin,95.09,79.59,0.00),v40,z0,tPen\WObj:=wPaper;
    MoveL Offs(pOrigin,95.51,80.22,0.00),v40,z0,tPen\WObj:=wPaper;
    MoveL Offs(pOrigin,95.09,79.59,0.00),v40,z0,tPen\WObj:=wPaper;
    MoveL Offs(pOrigin,95.93,79.79,0.00),v40,z0,tPen\WObj:=wPaper;
    MoveL Offs(pOrigin,89.62,73.48,0.00),v40,z0,tPen\WObj:=wPaper;
    MoveL Offs(pOrigin,89.34,73.69,0.00),v40,z0,tPen\WObj:=wPaper;
    MoveL Offs(pOrigin,94.60,68.43,0.00),v40,z0,tPen\WObj:=wPaper;
    MoveL Offs(pOrigin,94.40,69.30,0.00),v40,z0,tPen\WObj:=wPaper;
    MoveL Offs(pOrigin,93.49,68.40,0.00),v40,z0,tPen\WObj:=wPaper;
    MoveL Offs(pOrigin,93.85,67.69,0.00),v40,z0,tPen\WObj:=wPaper;
    MoveL Offs(pOrigin,89.04,72.49,0.00),v40,z0,tPen\WObj:=wPaper;
    MoveL Offs(pOrigin,89.78,72.02,0.00),v40,z0,tPen\WObj:=wPaper;
    MoveL Offs(pOrigin,91.48,72.02,0.00),v40,z0,tPen\WObj:=wPaper;
    MoveL Offs(pOrigin,90.83,72.36,0.00),v40,z0,tPen\WObj:=wPaper;
  ENDPROC

  PROC DrawPart280()
    MoveL Offs(pOrigin,90.83,73.42,0.00),v40,z0,tPen\WObj:=wPaper;
    MoveL Offs(pOrigin,90.20,73.08,0.00),v40,z0,tPen\WObj:=wPaper;
    MoveL Offs(pOrigin,91.69,73.08,0.00),v40,z0,tPen\WObj:=wPaper;
    MoveL Offs(pOrigin,92.31,73.19,0.00),v40,z0,tPen\WObj:=wPaper;
    MoveL Offs(pOrigin,88.85,69.73,0.00),v40,z0,tPen\WObj:=wPaper;
    MoveL Offs(pOrigin,89.35,69.91,0.00),v40,z0,tPen\WObj:=wPaper;
    MoveL Offs(pOrigin,90.84,69.91,0.00),v40,z0,tPen\WObj:=wPaper;
    MoveL Offs(pOrigin,91.25,69.14,0.00),v40,z0,tPen\WObj:=wPaper;
    MoveL Offs(pOrigin,88.85,66.74,0.00),v40,z0,tPen\WObj:=wPaper;
    MoveL Offs(pOrigin,89.14,66.74,0.00),v40,z0,tPen\WObj:=wPaper;
    MoveL Offs(pOrigin,90.84,66.74,0.00),v40,z0,tPen\WObj:=wPaper;
    MoveL Offs(pOrigin,91.24,66.15,0.00),v40,z0,tPen\WObj:=wPaper;
    MoveL Offs(pOrigin,88.99,63.89,0.00),v40,z0,tPen\WObj:=wPaper;
    MoveL Offs(pOrigin,88.62,63.96,0.00),v40,z0,tPen\WObj:=wPaper;
    MoveL Offs(pOrigin,96.88,55.69,0.00),v40,z0,tPen\WObj:=wPaper;
    MoveL Offs(pOrigin,96.29,54.80,0.00),v40,z0,tPen\WObj:=wPaper;
    MoveL Offs(pOrigin,88.47,62.61,0.00),v40,fine,tPen\WObj:=wPaper;
    MoveL Offs(pOrigin,88.47,62.61,6.00),v60,z5,tPen\WObj:=wPaper;
    MoveL Offs(pOrigin,89.56,63.58,6.00),vTravel,z5,tPen\WObj:=wPaper;
    MoveL Offs(pOrigin,89.56,63.58,0.00),v60,z0,tPen\WObj:=wPaper;
    MoveL Offs(pOrigin,91.05,63.58,0.00),v40,z0,tPen\WObj:=wPaper;
    MoveL Offs(pOrigin,91.38,63.30,0.00),v40,z0,tPen\WObj:=wPaper;
    MoveL Offs(pOrigin,89.43,61.35,0.00),v40,z0,tPen\WObj:=wPaper;
    MoveL Offs(pOrigin,89.99,61.46,0.00),v40,z0,tPen\WObj:=wPaper;
    MoveL Offs(pOrigin,91.48,61.46,0.00),v40,z0,tPen\WObj:=wPaper;
    MoveL Offs(pOrigin,90.83,61.74,0.00),v40,z0,tPen\WObj:=wPaper;
    MoveL Offs(pOrigin,90.83,60.46,0.00),v40,fine,tPen\WObj:=wPaper;
    MoveL Offs(pOrigin,90.83,60.46,6.00),v60,z5,tPen\WObj:=wPaper;
    MoveL Offs(pOrigin,88.93,60.66,6.00),vTravel,z5,tPen\WObj:=wPaper;
    MoveL Offs(pOrigin,88.93,60.66,0.00),v60,z0,tPen\WObj:=wPaper;
    MoveL Offs(pOrigin,95.84,53.75,0.00),v40,z0,tPen\WObj:=wPaper;
    MoveL Offs(pOrigin,95.40,53.88,0.00),v40,z0,tPen\WObj:=wPaper;
    MoveL Offs(pOrigin,91.94,50.42,0.00),v40,z0,tPen\WObj:=wPaper;
    MoveL Offs(pOrigin,92.32,50.90,0.00),v40,z0,tPen\WObj:=wPaper;
    MoveL Offs(pOrigin,94.45,50.90,0.00),v40,z0,tPen\WObj:=wPaper;
    MoveL Offs(pOrigin,94.00,50.90,0.00),v40,z0,tPen\WObj:=wPaper;
    MoveL Offs(pOrigin,94.00,56.85,0.00),v40,z0,tPen\WObj:=wPaper;
    MoveL Offs(pOrigin,93.18,56.85,0.00),v40,z0,tPen\WObj:=wPaper;
    MoveL Offs(pOrigin,95.44,61.74,0.00),v40,z0,tPen\WObj:=wPaper;
    MoveL Offs(pOrigin,96.36,62.38,0.00),v40,z0,tPen\WObj:=wPaper;
    MoveL Offs(pOrigin,96.36,62.38,0.00),v40,z0,tPen\WObj:=wPaper;
    MoveL Offs(pOrigin,98.91,67.69,0.00),v40,z0,tPen\WObj:=wPaper;
    MoveL Offs(pOrigin,98.50,67.52,0.00),v40,z0,tPen\WObj:=wPaper;
    MoveL Offs(pOrigin,101.50,64.52,0.00),v40,z0,tPen\WObj:=wPaper;
    MoveL Offs(pOrigin,100.75,63.77,0.00),v40,z0,tPen\WObj:=wPaper;
    MoveL Offs(pOrigin,97.75,66.78,0.00),v40,z0,tPen\WObj:=wPaper;
    MoveL Offs(pOrigin,97.00,66.03,0.00),v40,z0,tPen\WObj:=wPaper;
    MoveL Offs(pOrigin,100.16,62.87,0.00),v40,z0,tPen\WObj:=wPaper;
    MoveL Offs(pOrigin,99.71,61.83,0.00),v40,z0,tPen\WObj:=wPaper;
    MoveL Offs(pOrigin,96.56,64.98,0.00),v40,z0,tPen\WObj:=wPaper;
    MoveL Offs(pOrigin,95.81,64.23,0.00),v40,z0,tPen\WObj:=wPaper;
    MoveL Offs(pOrigin,99.12,60.93,0.00),v40,z0,tPen\WObj:=wPaper;
    MoveL Offs(pOrigin,98.67,59.88,0.00),v40,z0,tPen\WObj:=wPaper;
    MoveL Offs(pOrigin,95.36,63.19,0.00),v40,z0,tPen\WObj:=wPaper;
    MoveL Offs(pOrigin,95.58,63.01,0.00),v40,z0,tPen\WObj:=wPaper;
    MoveL Offs(pOrigin,102.49,69.93,0.00),v40,z0,tPen\WObj:=wPaper;
    MoveL Offs(pOrigin,103.28,70.20,0.00),v40,z0,tPen\WObj:=wPaper;
    MoveL Offs(pOrigin,101.63,71.86,0.00),v40,z0,tPen\WObj:=wPaper;
    MoveL Offs(pOrigin,102.22,72.75,0.00),v40,z0,tPen\WObj:=wPaper;
    MoveL Offs(pOrigin,103.73,71.25,0.00),v40,z0,tPen\WObj:=wPaper;
    MoveL Offs(pOrigin,104.17,72.30,0.00),v40,z0,tPen\WObj:=wPaper;
    MoveL Offs(pOrigin,102.67,73.80,0.00),v40,z0,tPen\WObj:=wPaper;
    MoveL Offs(pOrigin,103.25,73.67,0.00),v40,z0,tPen\WObj:=wPaper;
    MoveL Offs(pOrigin,105.65,76.08,0.00),v40,z0,tPen\WObj:=wPaper;
    MoveL Offs(pOrigin,105.50,75.97,0.00),v40,z0,tPen\WObj:=wPaper;
    MoveL Offs(pOrigin,105.71,76.40,0.00),v40,z0,tPen\WObj:=wPaper;
    MoveL Offs(pOrigin,105.50,75.97,0.00),v40,z0,tPen\WObj:=wPaper;
    MoveL Offs(pOrigin,106.56,75.89,0.00),v40,z0,tPen\WObj:=wPaper;
    MoveL Offs(pOrigin,105.21,77.24,0.00),v40,z0,tPen\WObj:=wPaper;
    MoveL Offs(pOrigin,106.14,77.04,0.00),v40,z0,tPen\WObj:=wPaper;
    MoveL Offs(pOrigin,106.56,77.46,0.00),v40,z0,tPen\WObj:=wPaper;
    MoveL Offs(pOrigin,106.14,77.04,0.00),v40,z0,tPen\WObj:=wPaper;
    MoveL Offs(pOrigin,107.16,76.78,0.00),v40,z0,tPen\WObj:=wPaper;
    MoveL Offs(pOrigin,105.65,78.29,0.00),v40,fine,tPen\WObj:=wPaper;
    MoveL Offs(pOrigin,105.65,78.29,6.00),v60,z5,tPen\WObj:=wPaper;
    MoveL Offs(pOrigin,104.75,79.19,6.00),vTravel,z5,tPen\WObj:=wPaper;
    MoveL Offs(pOrigin,104.75,79.19,0.00),v60,z0,tPen\WObj:=wPaper;
    MoveL Offs(pOrigin,100.54,83.39,0.00),v40,z0,tPen\WObj:=wPaper;
    MoveL Offs(pOrigin,99.80,82.65,0.00),v40,z0,tPen\WObj:=wPaper;
    MoveL Offs(pOrigin,103.85,78.59,0.00),v40,z0,tPen\WObj:=wPaper;
    MoveL Offs(pOrigin,103.11,77.84,0.00),v40,z0,tPen\WObj:=wPaper;
    MoveL Offs(pOrigin,99.05,81.90,0.00),v40,fine,tPen\WObj:=wPaper;
    MoveL Offs(pOrigin,99.05,81.90,6.00),v60,z5,tPen\WObj:=wPaper;
    MoveL Offs(pOrigin,100.40,81.50,6.00),vTravel,z5,tPen\WObj:=wPaper;
    MoveL Offs(pOrigin,100.40,81.50,0.00),v60,z0,tPen\WObj:=wPaper;
    MoveL Offs(pOrigin,101.46,81.78,0.00),v40,z0,tPen\WObj:=wPaper;
    MoveL Offs(pOrigin,107.20,85.82,0.00),v40,z0,tPen\WObj:=wPaper;
    MoveL Offs(pOrigin,112.02,88.37,0.00),v40,z0,tPen\WObj:=wPaper;
    MoveL Offs(pOrigin,112.51,89.08,0.00),v40,z0,tPen\WObj:=wPaper;
    MoveL Offs(pOrigin,117.82,90.85,0.00),v40,z0,tPen\WObj:=wPaper;
    MoveL Offs(pOrigin,117.15,90.68,0.00),v40,z0,tPen\WObj:=wPaper;
    MoveL Offs(pOrigin,113.39,94.44,0.00),v40,z0,tPen\WObj:=wPaper;
    MoveL Offs(pOrigin,113.05,93.93,0.00),v40,z0,tPen\WObj:=wPaper;
    MoveL Offs(pOrigin,110.79,91.67,0.00),v40,z0,tPen\WObj:=wPaper;
    MoveL Offs(pOrigin,110.56,91.30,0.00),v40,z0,tPen\WObj:=wPaper;
    MoveL Offs(pOrigin,108.90,92.96,0.00),v40,z0,tPen\WObj:=wPaper;
    MoveL Offs(pOrigin,108.90,91.91,0.00),v40,z0,tPen\WObj:=wPaper;
    MoveL Offs(pOrigin,109.54,91.70,0.00),v40,z0,tPen\WObj:=wPaper;
    MoveL Offs(pOrigin,115.28,92.76,0.00),v40,z0,tPen\WObj:=wPaper;
    MoveL Offs(pOrigin,119.74,92.76,0.00),v40,z0,tPen\WObj:=wPaper;
    MoveL Offs(pOrigin,125.05,91.91,0.00),v40,z0,tPen\WObj:=wPaper;
    MoveL Offs(pOrigin,128.02,90.99,0.00),v40,z0,tPen\WObj:=wPaper;
    MoveL Offs(pOrigin,128.45,90.43,0.00),v40,z0,tPen\WObj:=wPaper;
    MoveL Offs(pOrigin,128.01,89.48,0.00),v40,z0,tPen\WObj:=wPaper;
    MoveL Offs(pOrigin,130.57,92.03,0.00),v40,z0,tPen\WObj:=wPaper;
    MoveL Offs(pOrigin,130.03,92.74,0.00),v40,z0,tPen\WObj:=wPaper;
    MoveL Offs(pOrigin,142.05,80.72,0.00),v40,z0,tPen\WObj:=wPaper;
    MoveL Offs(pOrigin,142.22,81.28,0.00),v40,z0,tPen\WObj:=wPaper;
    MoveL Offs(pOrigin,145.07,84.14,0.00),v40,z0,tPen\WObj:=wPaper;
    MoveL Offs(pOrigin,145.82,83.39,0.00),v40,z0,tPen\WObj:=wPaper;
    MoveL Offs(pOrigin,143.42,80.99,0.00),v40,z0,tPen\WObj:=wPaper;
    MoveL Offs(pOrigin,143.63,81.71,0.00),v40,z0,tPen\WObj:=wPaper;
    MoveL Offs(pOrigin,143.63,83.84,0.00),v40,z0,tPen\WObj:=wPaper;
    MoveL Offs(pOrigin,144.03,84.58,0.00),v40,z0,tPen\WObj:=wPaper;
    MoveL Offs(pOrigin,141.17,81.73,0.00),v40,z0,tPen\WObj:=wPaper;
    MoveL Offs(pOrigin,141.52,82.78,0.00),v40,z0,tPen\WObj:=wPaper;
    MoveL Offs(pOrigin,141.52,85.11,0.00),v40,fine,tPen\WObj:=wPaper;
    MoveL Offs(pOrigin,141.52,85.11,6.00),v60,z5,tPen\WObj:=wPaper;
    MoveL Offs(pOrigin,142.57,84.48,6.00),vTravel,z5,tPen\WObj:=wPaper;
    MoveL Offs(pOrigin,142.57,84.48,0.00),v60,z0,tPen\WObj:=wPaper;
  ENDPROC

  PROC DrawPart281()
    MoveL Offs(pOrigin,142.57,82.14,0.00),v40,z0,tPen\WObj:=wPaper;
    MoveL Offs(pOrigin,142.48,81.53,0.00),v40,z0,tPen\WObj:=wPaper;
    MoveL Offs(pOrigin,147.79,81.53,0.00),v40,z0,tPen\WObj:=wPaper;
    MoveL Offs(pOrigin,147.36,81.93,0.00),v40,z0,tPen\WObj:=wPaper;
    MoveL Offs(pOrigin,139.07,87.52,0.00),v40,z0,tPen\WObj:=wPaper;
    MoveL Offs(pOrigin,133.34,90.50,0.00),v40,z0,tPen\WObj:=wPaper;
    MoveL Offs(pOrigin,128.02,92.55,0.00),v40,z0,tPen\WObj:=wPaper;
    MoveL Offs(pOrigin,123.78,93.61,0.00),v40,z0,tPen\WObj:=wPaper;
    MoveL Offs(pOrigin,120.38,94.04,0.00),v40,z0,tPen\WObj:=wPaper;
    MoveL Offs(pOrigin,114.21,93.82,0.00),v40,z0,tPen\WObj:=wPaper;
    MoveL Offs(pOrigin,109.11,92.48,0.00),v40,z0,tPen\WObj:=wPaper;
    MoveL Offs(pOrigin,108.47,91.77,0.00),v40,z0,tPen\WObj:=wPaper;
    MoveL Offs(pOrigin,105.50,90.64,0.00),v40,z0,tPen\WObj:=wPaper;
    MoveL Offs(pOrigin,106.06,91.32,0.00),v40,z0,tPen\WObj:=wPaper;
    MoveL Offs(pOrigin,107.11,90.26,0.00),v40,fine,tPen\WObj:=wPaper;
    MoveL Offs(pOrigin,107.11,90.26,6.00),v60,z5,tPen\WObj:=wPaper;
    MoveL Offs(pOrigin,108.46,90.41,6.00),vTravel,z5,tPen\WObj:=wPaper;
    MoveL Offs(pOrigin,108.46,90.41,0.00),v60,z0,tPen\WObj:=wPaper;
    MoveL Offs(pOrigin,106.81,92.06,0.00),v40,z0,tPen\WObj:=wPaper;
    MoveL Offs(pOrigin,107.71,92.66,0.00),v40,z0,tPen\WObj:=wPaper;
    MoveL Offs(pOrigin,109.51,90.86,0.00),v40,z0,tPen\WObj:=wPaper;
    MoveL Offs(pOrigin,109.14,91.52,0.00),v40,z0,tPen\WObj:=wPaper;
    MoveL Offs(pOrigin,111.10,93.47,0.00),v40,z0,tPen\WObj:=wPaper;
    MoveL Offs(pOrigin,111.00,93.85,0.00),v40,z0,tPen\WObj:=wPaper;
    MoveL Offs(pOrigin,113.40,91.44,0.00),v40,z0,tPen\WObj:=wPaper;
    MoveL Offs(pOrigin,112.74,92.13,0.00),v40,z0,tPen\WObj:=wPaper;
    MoveL Offs(pOrigin,114.70,94.08,0.00),v40,z0,tPen\WObj:=wPaper;
    MoveL Offs(pOrigin,114.59,94.74,0.00),v40,z0,tPen\WObj:=wPaper;
    MoveL Offs(pOrigin,117.75,91.58,0.00),v40,z0,tPen\WObj:=wPaper;
    MoveL Offs(pOrigin,117.54,92.44,0.00),v40,z0,tPen\WObj:=wPaper;
    MoveL Offs(pOrigin,119.49,94.39,0.00),v40,z0,tPen\WObj:=wPaper;
    MoveL Offs(pOrigin,118.93,94.87,0.00),v40,z0,tPen\WObj:=wPaper;
    MoveL Offs(pOrigin,125.40,88.41,0.00),v40,fine,tPen\WObj:=wPaper;
    MoveL Offs(pOrigin,125.40,88.41,6.00),v60,z5,tPen\WObj:=wPaper;
    MoveL Offs(pOrigin,126.59,88.71,6.00),vTravel,z5,tPen\WObj:=wPaper;
    MoveL Offs(pOrigin,126.59,88.71,0.00),v60,z0,tPen\WObj:=wPaper;
    MoveL Offs(pOrigin,120.58,94.72,0.00),v40,z0,tPen\WObj:=wPaper;
    MoveL Offs(pOrigin,120.99,94.40,0.00),v40,z0,tPen\WObj:=wPaper;
    MoveL Offs(pOrigin,119.03,92.45,0.00),v40,z0,tPen\WObj:=wPaper;
    MoveL Offs(pOrigin,118.94,91.88,0.00),v40,z0,tPen\WObj:=wPaper;
    MoveL Offs(pOrigin,116.09,94.73,0.00),v40,z0,tPen\WObj:=wPaper;
    MoveL Offs(pOrigin,116.49,94.39,0.00),v40,z0,tPen\WObj:=wPaper;
    MoveL Offs(pOrigin,114.54,92.43,0.00),v40,fine,tPen\WObj:=wPaper;
    MoveL Offs(pOrigin,114.54,92.43,6.00),v60,z5,tPen\WObj:=wPaper;
    MoveL Offs(pOrigin,116.04,92.44,6.00),vTravel,z5,tPen\WObj:=wPaper;
    MoveL Offs(pOrigin,116.04,92.44,0.00),v60,z0,tPen\WObj:=wPaper;
    MoveL Offs(pOrigin,118.14,94.54,0.00),v40,z0,tPen\WObj:=wPaper;
    MoveL Offs(pOrigin,117.44,94.88,0.00),v40,z0,tPen\WObj:=wPaper;
    MoveL Offs(pOrigin,120.74,91.57,0.00),v40,z0,tPen\WObj:=wPaper;
    MoveL Offs(pOrigin,120.53,92.45,0.00),v40,z0,tPen\WObj:=wPaper;
    MoveL Offs(pOrigin,122.19,94.10,0.00),v40,z0,tPen\WObj:=wPaper;
    MoveL Offs(pOrigin,122.08,94.71,0.00),v40,z0,tPen\WObj:=wPaper;
    MoveL Offs(pOrigin,128.09,88.70,0.00),v40,fine,tPen\WObj:=wPaper;
    MoveL Offs(pOrigin,128.09,88.70,6.00),v60,z5,tPen\WObj:=wPaper;
    MoveL Offs(pOrigin,129.59,88.70,6.00),vTravel,z5,tPen\WObj:=wPaper;
    MoveL Offs(pOrigin,129.59,88.70,0.00),v60,z0,tPen\WObj:=wPaper;
    MoveL Offs(pOrigin,124.03,94.26,0.00),v40,z0,tPen\WObj:=wPaper;
    MoveL Offs(pOrigin,123.53,93.96,0.00),v40,z0,tPen\WObj:=wPaper;
    MoveL Offs(pOrigin,121.73,92.15,0.00),v40,fine,tPen\WObj:=wPaper;
    MoveL Offs(pOrigin,121.73,92.15,6.00),v60,z5,tPen\WObj:=wPaper;
    MoveL Offs(pOrigin,123.08,92.01,6.00),vTravel,z5,tPen\WObj:=wPaper;
    MoveL Offs(pOrigin,123.08,92.01,0.00),v60,z0,tPen\WObj:=wPaper;
    MoveL Offs(pOrigin,124.88,93.81,0.00),v40,z0,tPen\WObj:=wPaper;
    MoveL Offs(pOrigin,125.05,93.14,0.00),v40,z0,tPen\WObj:=wPaper;
    MoveL Offs(pOrigin,112.94,93.14,0.00),v40,fine,tPen\WObj:=wPaper;
    MoveL Offs(pOrigin,112.94,93.14,6.00),v60,z5,tPen\WObj:=wPaper;
    MoveL Offs(pOrigin,112.05,94.29,6.00),vTravel,z5,tPen\WObj:=wPaper;
    MoveL Offs(pOrigin,112.05,94.29,0.00),v60,z0,tPen\WObj:=wPaper;
    MoveL Offs(pOrigin,116.55,89.79,0.00),v40,z0,tPen\WObj:=wPaper;
    MoveL Offs(pOrigin,115.81,89.04,0.00),v40,z0,tPen\WObj:=wPaper;
    MoveL Offs(pOrigin,114.15,90.69,0.00),v40,z0,tPen\WObj:=wPaper;
    MoveL Offs(pOrigin,113.48,89.88,0.00),v40,z0,tPen\WObj:=wPaper;
    MoveL Offs(pOrigin,111.53,87.93,0.00),v40,z0,tPen\WObj:=wPaper;
    MoveL Offs(pOrigin,111.62,87.26,0.00),v40,z0,tPen\WObj:=wPaper;
    MoveL Offs(pOrigin,109.81,89.06,0.00),v40,z0,tPen\WObj:=wPaper;
    MoveL Offs(pOrigin,109.29,88.67,0.00),v40,z0,tPen\WObj:=wPaper;
    MoveL Offs(pOrigin,103.58,82.96,0.00),v40,z0,tPen\WObj:=wPaper;
    MoveL Offs(pOrigin,103.80,83.64,0.00),v40,z0,tPen\WObj:=wPaper;
    MoveL Offs(pOrigin,102.74,83.64,0.00),v40,z0,tPen\WObj:=wPaper;
    MoveL Offs(pOrigin,101.78,84.15,0.00),v40,z0,tPen\WObj:=wPaper;
    MoveL Offs(pOrigin,98.18,80.55,0.00),v40,fine,tPen\WObj:=wPaper;
    MoveL Offs(pOrigin,98.18,80.55,6.00),v60,z5,tPen\WObj:=wPaper;
    MoveL Offs(pOrigin,97.87,78.75,6.00),vTravel,z5,tPen\WObj:=wPaper;
    MoveL Offs(pOrigin,97.87,78.75,0.00),v60,z0,tPen\WObj:=wPaper;
    MoveL Offs(pOrigin,105.98,86.86,0.00),v40,z0,tPen\WObj:=wPaper;
    MoveL Offs(pOrigin,105.78,87.12,0.00),v40,z0,tPen\WObj:=wPaper;
    MoveL Offs(pOrigin,107.73,85.17,0.00),v40,z0,tPen\WObj:=wPaper;
    MoveL Offs(pOrigin,108.08,85.97,0.00),v40,z0,tPen\WObj:=wPaper;
    MoveL Offs(pOrigin,111.54,89.43,0.00),v40,z0,tPen\WObj:=wPaper;
    MoveL Offs(pOrigin,111.76,90.10,0.00),v40,z0,tPen\WObj:=wPaper;
    MoveL Offs(pOrigin,113.56,88.30,0.00),v40,z0,tPen\WObj:=wPaper;
    MoveL Offs(pOrigin,112.66,87.70,0.00),v40,z0,tPen\WObj:=wPaper;
    MoveL Offs(pOrigin,110.71,89.65,0.00),v40,fine,tPen\WObj:=wPaper;
    MoveL Offs(pOrigin,110.71,89.65,6.00),v60,z5,tPen\WObj:=wPaper;
    MoveL Offs(pOrigin,112.09,88.72,6.00),vTravel,z5,tPen\WObj:=wPaper;
    MoveL Offs(pOrigin,112.09,88.72,0.00),v60,z0,tPen\WObj:=wPaper;
    MoveL Offs(pOrigin,112.30,89.15,0.00),v40,z0,tPen\WObj:=wPaper;
    MoveL Offs(pOrigin,112.09,88.72,0.00),v40,z0,tPen\WObj:=wPaper;
    MoveL Offs(pOrigin,112.30,89.15,0.00),v40,z0,tPen\WObj:=wPaper;
    MoveL Offs(pOrigin,111.24,89.01,0.00),v40,z0,tPen\WObj:=wPaper;
    MoveL Offs(pOrigin,108.26,87.73,0.00),v40,z0,tPen\WObj:=wPaper;
    MoveL Offs(pOrigin,103.59,84.90,0.00),v40,z0,tPen\WObj:=wPaper;
    MoveL Offs(pOrigin,100.82,82.78,0.00),v40,z0,tPen\WObj:=wPaper;
    MoveL Offs(pOrigin,100.19,81.50,0.00),v40,z0,tPen\WObj:=wPaper;
    MoveL Offs(pOrigin,95.72,76.82,0.00),v40,z0,tPen\WObj:=wPaper;
    MoveL Offs(pOrigin,94.87,77.12,0.00),v40,z0,tPen\WObj:=wPaper;
    MoveL Offs(pOrigin,92.47,79.52,0.00),v40,z0,tPen\WObj:=wPaper;
    MoveL Offs(pOrigin,92.63,79.48,0.00),v40,z0,tPen\WObj:=wPaper;
    MoveL Offs(pOrigin,98.49,85.34,0.00),v40,z0,tPen\WObj:=wPaper;
    MoveL Offs(pOrigin,98.89,85.05,0.00),v40,z0,tPen\WObj:=wPaper;
    MoveL Offs(pOrigin,96.19,87.75,0.00),v40,z0,tPen\WObj:=wPaper;
    MoveL Offs(pOrigin,96.78,88.65,0.00),v40,z0,tPen\WObj:=wPaper;
    MoveL Offs(pOrigin,99.34,86.09,0.00),v40,z0,tPen\WObj:=wPaper;
    MoveL Offs(pOrigin,98.49,86.81,0.00),v40,z0,tPen\WObj:=wPaper;
    MoveL Offs(pOrigin,97.00,86.81,0.00),v40,z0,tPen\WObj:=wPaper;
    MoveL Offs(pOrigin,97.43,87.86,0.00),v40,z0,tPen\WObj:=wPaper;
    MoveL Offs(pOrigin,98.91,87.86,0.00),v40,fine,tPen\WObj:=wPaper;
    MoveL Offs(pOrigin,98.91,87.86,6.00),v60,z5,tPen\WObj:=wPaper;
    MoveL Offs(pOrigin,97.64,88.72,6.00),vTravel,z5,tPen\WObj:=wPaper;
    MoveL Offs(pOrigin,97.64,88.72,0.00),v60,z0,tPen\WObj:=wPaper;
  ENDPROC

  PROC DrawPart282()
    MoveL Offs(pOrigin,97.85,89.15,0.00),v40,z0,tPen\WObj:=wPaper;
    MoveL Offs(pOrigin,97.64,88.72,0.00),v40,z0,tPen\WObj:=wPaper;
    MoveL Offs(pOrigin,97.15,88.48,0.00),v40,z0,tPen\WObj:=wPaper;
    MoveL Offs(pOrigin,105.87,97.20,0.00),v40,z0,tPen\WObj:=wPaper;
    MoveL Offs(pOrigin,105.29,97.37,0.00),v40,z0,tPen\WObj:=wPaper;
    MoveL Offs(pOrigin,104.01,97.37,0.00),v40,z0,tPen\WObj:=wPaper;
    MoveL Offs(pOrigin,104.22,98.42,0.00),v40,z0,tPen\WObj:=wPaper;
    MoveL Offs(pOrigin,105.71,98.42,0.00),v40,z0,tPen\WObj:=wPaper;
    MoveL Offs(pOrigin,105.93,99.48,0.00),v40,z0,tPen\WObj:=wPaper;
    MoveL Offs(pOrigin,104.44,99.48,0.00),v40,fine,tPen\WObj:=wPaper;
    MoveL Offs(pOrigin,104.44,99.48,6.00),v60,z5,tPen\WObj:=wPaper;
    MoveL Offs(pOrigin,102.90,97.47,6.00),vTravel,z5,tPen\WObj:=wPaper;
    MoveL Offs(pOrigin,102.90,97.47,0.00),v60,z0,tPen\WObj:=wPaper;
    MoveL Offs(pOrigin,106.65,93.71,0.00),v40,z0,tPen\WObj:=wPaper;
    MoveL Offs(pOrigin,105.61,93.27,0.00),v40,z0,tPen\WObj:=wPaper;
    MoveL Offs(pOrigin,102.60,96.27,0.00),v40,z0,tPen\WObj:=wPaper;
    MoveL Offs(pOrigin,103.59,96.31,0.00),v40,z0,tPen\WObj:=wPaper;
    MoveL Offs(pOrigin,105.29,96.31,0.00),v40,z0,tPen\WObj:=wPaper;
    MoveL Offs(pOrigin,104.56,96.16,0.00),v40,z0,tPen\WObj:=wPaper;
    MoveL Offs(pOrigin,104.56,94.25,0.00),v40,z0,tPen\WObj:=wPaper;
    MoveL Offs(pOrigin,105.50,94.20,0.00),v40,z0,tPen\WObj:=wPaper;
    MoveL Offs(pOrigin,102.52,94.20,0.00),v40,z0,tPen\WObj:=wPaper;
    MoveL Offs(pOrigin,101.89,93.61,0.00),v40,z0,tPen\WObj:=wPaper;
    MoveL Offs(pOrigin,102.31,94.04,0.00),v40,z0,tPen\WObj:=wPaper;
    MoveL Offs(pOrigin,101.89,93.61,0.00),v40,z0,tPen\WObj:=wPaper;
    MoveL Offs(pOrigin,101.56,94.33,0.00),v40,z0,tPen\WObj:=wPaper;
    MoveL Offs(pOrigin,103.96,91.92,0.00),v40,fine,tPen\WObj:=wPaper;
    MoveL Offs(pOrigin,103.96,91.92,6.00),v60,z5,tPen\WObj:=wPaper;
    MoveL Offs(pOrigin,101.57,89.83,6.00),vTravel,z5,tPen\WObj:=wPaper;
    MoveL Offs(pOrigin,101.57,89.83,0.00),v60,z0,tPen\WObj:=wPaper;
    MoveL Offs(pOrigin,99.17,92.24,0.00),v40,fine,tPen\WObj:=wPaper;
    MoveL Offs(pOrigin,99.17,92.24,6.00),v60,z5,tPen\WObj:=wPaper;
    MoveL Offs(pOrigin,100.40,90.00,6.00),vTravel,z5,tPen\WObj:=wPaper;
    MoveL Offs(pOrigin,100.40,90.00,0.00),v60,z0,tPen\WObj:=wPaper;
    MoveL Offs(pOrigin,101.89,91.70,0.00),v40,z0,tPen\WObj:=wPaper;
    MoveL Offs(pOrigin,100.40,90.00,0.00),v40,fine,tPen\WObj:=wPaper;
    MoveL Offs(pOrigin,100.40,90.00,6.00),v60,z5,tPen\WObj:=wPaper;
    MoveL Offs(pOrigin,98.06,85.75,6.00),vTravel,z5,tPen\WObj:=wPaper;
    MoveL Offs(pOrigin,98.06,85.75,0.00),v60,z0,tPen\WObj:=wPaper;
    MoveL Offs(pOrigin,96.58,85.75,0.00),v40,z0,tPen\WObj:=wPaper;
    MoveL Offs(pOrigin,96.36,84.70,0.00),v40,z0,tPen\WObj:=wPaper;
    MoveL Offs(pOrigin,97.85,84.70,0.00),v40,z0,tPen\WObj:=wPaper;
    MoveL Offs(pOrigin,98.45,84.00,0.00),v40,z0,tPen\WObj:=wPaper;
    MoveL Offs(pOrigin,95.74,86.70,0.00),v40,fine,tPen\WObj:=wPaper;
    MoveL Offs(pOrigin,95.74,86.70,6.00),v60,z5,tPen\WObj:=wPaper;
    MoveL Offs(pOrigin,101.29,84.14,6.00),vTravel,z5,tPen\WObj:=wPaper;
    MoveL Offs(pOrigin,101.29,84.14,0.00),v60,z0,tPen\WObj:=wPaper;
    MoveL Offs(pOrigin,105.50,79.93,0.00),v40,z0,tPen\WObj:=wPaper;
    MoveL Offs(pOrigin,106.24,80.68,0.00),v40,z0,tPen\WObj:=wPaper;
    MoveL Offs(pOrigin,102.19,84.74,0.00),v40,z0,tPen\WObj:=wPaper;
    MoveL Offs(pOrigin,103.08,85.33,0.00),v40,z0,tPen\WObj:=wPaper;
    MoveL Offs(pOrigin,105.19,83.23,0.00),v40,z0,tPen\WObj:=wPaper;
    MoveL Offs(pOrigin,105.94,83.98,0.00),v40,z0,tPen\WObj:=wPaper;
    MoveL Offs(pOrigin,103.83,86.08,0.00),v40,z0,tPen\WObj:=wPaper;
    MoveL Offs(pOrigin,104.88,86.53,0.00),v40,z0,tPen\WObj:=wPaper;
    MoveL Offs(pOrigin,106.83,84.57,0.00),v40,fine,tPen\WObj:=wPaper;
    MoveL Offs(pOrigin,106.83,84.57,6.00),v60,z5,tPen\WObj:=wPaper;
    MoveL Offs(pOrigin,105.29,84.70,6.00),vTravel,z5,tPen\WObj:=wPaper;
    MoveL Offs(pOrigin,105.29,84.70,0.00),v60,z0,tPen\WObj:=wPaper;
    MoveL Offs(pOrigin,104.22,84.70,0.00),v40,z0,tPen\WObj:=wPaper;
    MoveL Offs(pOrigin,104.22,84.05,0.00),v40,z0,tPen\WObj:=wPaper;
    MoveL Offs(pOrigin,104.86,84.47,0.00),v40,z0,tPen\WObj:=wPaper;
    MoveL Offs(pOrigin,104.22,84.05,0.00),v40,fine,tPen\WObj:=wPaper;
    MoveL Offs(pOrigin,104.22,84.05,6.00),v60,z5,tPen\WObj:=wPaper;
    MoveL Offs(pOrigin,102.31,82.56,6.00),vTravel,z5,tPen\WObj:=wPaper;
    MoveL Offs(pOrigin,102.31,82.56,0.00),v60,z0,tPen\WObj:=wPaper;
    MoveL Offs(pOrigin,102.74,82.99,0.00),v40,z0,tPen\WObj:=wPaper;
    MoveL Offs(pOrigin,102.31,82.56,0.00),v40,fine,tPen\WObj:=wPaper;
    MoveL Offs(pOrigin,102.31,82.56,6.00),v60,z5,tPen\WObj:=wPaper;
    MoveL Offs(pOrigin,104.32,80.72,6.00),vTravel,z5,tPen\WObj:=wPaper;
    MoveL Offs(pOrigin,104.32,80.72,0.00),v60,z0,tPen\WObj:=wPaper;
    MoveL Offs(pOrigin,93.05,69.45,0.00),v40,fine,tPen\WObj:=wPaper;
    MoveL Offs(pOrigin,93.05,69.45,6.00),v60,z5,tPen\WObj:=wPaper;
    MoveL Offs(pOrigin,94.24,70.45,6.00),vTravel,z5,tPen\WObj:=wPaper;
    MoveL Offs(pOrigin,94.24,70.45,0.00),v60,z0,tPen\WObj:=wPaper;
    MoveL Offs(pOrigin,94.45,70.88,0.00),v40,z0,tPen\WObj:=wPaper;
    MoveL Offs(pOrigin,94.24,70.45,0.00),v40,z0,tPen\WObj:=wPaper;
    MoveL Offs(pOrigin,94.45,70.88,0.00),v40,z0,tPen\WObj:=wPaper;
    MoveL Offs(pOrigin,94.80,71.94,0.00),v40,z0,tPen\WObj:=wPaper;
    MoveL Offs(pOrigin,96.79,74.49,0.00),v40,z0,tPen\WObj:=wPaper;
    MoveL Offs(pOrigin,99.97,77.46,0.00),v40,z0,tPen\WObj:=wPaper;
    MoveL Offs(pOrigin,101.04,77.89,0.00),v40,z0,tPen\WObj:=wPaper;
    MoveL Offs(pOrigin,101.04,77.89,0.00),v40,z0,tPen\WObj:=wPaper;
    MoveL Offs(pOrigin,107.41,82.56,0.00),v40,fine,tPen\WObj:=wPaper;
    MoveL Offs(pOrigin,107.41,82.56,6.00),v60,z5,tPen\WObj:=wPaper;
    MoveL Offs(pOrigin,108.34,81.57,6.00),vTravel,z5,tPen\WObj:=wPaper;
    MoveL Offs(pOrigin,108.34,81.57,0.00),v60,z0,tPen\WObj:=wPaper;
    MoveL Offs(pOrigin,109.84,80.07,0.00),v40,z0,tPen\WObj:=wPaper;
    MoveL Offs(pOrigin,110.44,80.97,0.00),v40,z0,tPen\WObj:=wPaper;
    MoveL Offs(pOrigin,109.09,82.32,0.00),v40,z0,tPen\WObj:=wPaper;
    MoveL Offs(pOrigin,109.83,83.07,0.00),v40,z0,tPen\WObj:=wPaper;
    MoveL Offs(pOrigin,111.34,81.56,0.00),v40,z0,tPen\WObj:=wPaper;
    MoveL Offs(pOrigin,112.23,82.16,0.00),v40,z0,tPen\WObj:=wPaper;
    MoveL Offs(pOrigin,110.58,83.81,0.00),v40,z0,tPen\WObj:=wPaper;
    MoveL Offs(pOrigin,111.48,84.41,0.00),v40,z0,tPen\WObj:=wPaper;
    MoveL Offs(pOrigin,112.83,83.06,0.00),v40,z0,tPen\WObj:=wPaper;
    MoveL Offs(pOrigin,113.73,83.65,0.00),v40,z0,tPen\WObj:=wPaper;
    MoveL Offs(pOrigin,112.22,85.16,0.00),v40,z0,tPen\WObj:=wPaper;
    MoveL Offs(pOrigin,112.97,85.90,0.00),v40,z0,tPen\WObj:=wPaper;
    MoveL Offs(pOrigin,114.62,84.25,0.00),v40,fine,tPen\WObj:=wPaper;
    MoveL Offs(pOrigin,114.62,84.25,6.00),v60,z5,tPen\WObj:=wPaper;
    MoveL Offs(pOrigin,116.42,85.44,6.00),vTravel,z5,tPen\WObj:=wPaper;
    MoveL Offs(pOrigin,116.42,85.44,0.00),v60,z0,tPen\WObj:=wPaper;
    MoveL Offs(pOrigin,114.76,87.10,0.00),v40,z0,tPen\WObj:=wPaper;
    MoveL Offs(pOrigin,115.66,87.69,0.00),v40,z0,tPen\WObj:=wPaper;
    MoveL Offs(pOrigin,117.46,85.89,0.00),v40,z0,tPen\WObj:=wPaper;
    MoveL Offs(pOrigin,118.36,86.49,0.00),v40,z0,tPen\WObj:=wPaper;
    MoveL Offs(pOrigin,116.56,88.29,0.00),v40,z0,tPen\WObj:=wPaper;
    MoveL Offs(pOrigin,117.60,88.73,0.00),v40,z0,tPen\WObj:=wPaper;
    MoveL Offs(pOrigin,119.41,86.93,0.00),v40,fine,tPen\WObj:=wPaper;
    MoveL Offs(pOrigin,119.41,86.93,6.00),v60,z5,tPen\WObj:=wPaper;
    MoveL Offs(pOrigin,121.65,87.67,6.00),vTravel,z5,tPen\WObj:=wPaper;
    MoveL Offs(pOrigin,121.65,87.67,0.00),v60,z0,tPen\WObj:=wPaper;
    MoveL Offs(pOrigin,119.70,89.63,0.00),v40,fine,tPen\WObj:=wPaper;
    MoveL Offs(pOrigin,119.70,89.63,6.00),v60,z5,tPen\WObj:=wPaper;
    MoveL Offs(pOrigin,114.61,88.74,6.00),vTravel,z5,tPen\WObj:=wPaper;
    MoveL Offs(pOrigin,114.61,88.74,0.00),v60,z0,tPen\WObj:=wPaper;
    MoveL Offs(pOrigin,112.96,90.40,0.00),v40,fine,tPen\WObj:=wPaper;
    MoveL Offs(pOrigin,112.96,90.40,6.00),v60,z5,tPen\WObj:=wPaper;
    MoveL Offs(pOrigin,111.90,91.45,6.00),vTravel,z5,tPen\WObj:=wPaper;
  ENDPROC

  PROC DrawPart283()
    MoveL Offs(pOrigin,111.90,91.45,0.00),v60,z0,tPen\WObj:=wPaper;
    MoveL Offs(pOrigin,109.95,93.40,0.00),v40,fine,tPen\WObj:=wPaper;
    MoveL Offs(pOrigin,109.95,93.40,6.00),v60,z5,tPen\WObj:=wPaper;
    MoveL Offs(pOrigin,108.26,97.22,6.00),vTravel,z5,tPen\WObj:=wPaper;
    MoveL Offs(pOrigin,108.26,97.22,0.00),v60,z0,tPen\WObj:=wPaper;
    MoveL Offs(pOrigin,108.90,97.65,0.00),v40,z0,tPen\WObj:=wPaper;
    MoveL Offs(pOrigin,108.26,97.22,0.00),v40,fine,tPen\WObj:=wPaper;
    MoveL Offs(pOrigin,108.26,97.22,6.00),v60,z5,tPen\WObj:=wPaper;
    MoveL Offs(pOrigin,106.99,98.50,6.00),vTravel,z5,tPen\WObj:=wPaper;
    MoveL Offs(pOrigin,106.99,98.50,0.00),v60,z0,tPen\WObj:=wPaper;
    MoveL Offs(pOrigin,109.68,103.81,0.00),v40,z0,tPen\WObj:=wPaper;
    MoveL Offs(pOrigin,112.94,107.85,0.00),v40,z0,tPen\WObj:=wPaper;
    MoveL Offs(pOrigin,112.94,107.85,0.00),v40,z0,tPen\WObj:=wPaper;
    MoveL Offs(pOrigin,113.36,109.12,0.00),v40,z0,tPen\WObj:=wPaper;
    MoveL Offs(pOrigin,114.64,109.55,0.00),v40,z0,tPen\WObj:=wPaper;
    MoveL Offs(pOrigin,114.64,109.55,0.00),v40,z0,tPen\WObj:=wPaper;
    MoveL Offs(pOrigin,114.43,108.70,0.00),v40,z0,tPen\WObj:=wPaper;
    MoveL Offs(pOrigin,113.79,108.06,0.00),v40,z0,tPen\WObj:=wPaper;
    MoveL Offs(pOrigin,112.94,107.85,0.00),v40,z0,tPen\WObj:=wPaper;
    MoveL Offs(pOrigin,112.94,107.85,0.00),v40,z0,tPen\WObj:=wPaper;
    MoveL Offs(pOrigin,111.88,107.00,0.00),v40,z0,tPen\WObj:=wPaper;
    MoveL Offs(pOrigin,111.14,106.95,0.00),v40,z0,tPen\WObj:=wPaper;
    MoveL Offs(pOrigin,114.14,109.96,0.00),v40,z0,tPen\WObj:=wPaper;
    MoveL Offs(pOrigin,113.94,110.32,0.00),v40,z0,tPen\WObj:=wPaper;
    MoveL Offs(pOrigin,115.60,108.66,0.00),v40,z0,tPen\WObj:=wPaper;
    MoveL Offs(pOrigin,114.85,107.92,0.00),v40,z0,tPen\WObj:=wPaper;
    MoveL Offs(pOrigin,113.05,109.72,0.00),v40,fine,tPen\WObj:=wPaper;
    MoveL Offs(pOrigin,113.05,109.72,6.00),v60,z5,tPen\WObj:=wPaper;
    MoveL Offs(pOrigin,114.64,109.55,6.00),vTravel,z5,tPen\WObj:=wPaper;
    MoveL Offs(pOrigin,114.64,109.55,0.00),v60,z0,tPen\WObj:=wPaper;
    MoveL Offs(pOrigin,116.12,110.40,0.00),v40,z0,tPen\WObj:=wPaper;
    MoveL Offs(pOrigin,116.12,110.40,0.00),v40,z0,tPen\WObj:=wPaper;
    MoveL Offs(pOrigin,117.19,110.40,0.00),v40,z0,tPen\WObj:=wPaper;
    MoveL Offs(pOrigin,117.40,111.25,0.00),v40,z0,tPen\WObj:=wPaper;
    MoveL Offs(pOrigin,117.40,111.25,0.00),v40,z0,tPen\WObj:=wPaper;
    MoveL Offs(pOrigin,117.82,111.46,0.00),v40,z0,tPen\WObj:=wPaper;
    MoveL Offs(pOrigin,118.04,112.10,0.00),v40,z0,tPen\WObj:=wPaper;
    MoveL Offs(pOrigin,119.10,112.10,0.00),v40,z0,tPen\WObj:=wPaper;
    MoveL Offs(pOrigin,118.58,113.15,0.00),v40,z0,tPen\WObj:=wPaper;
    MoveL Offs(pOrigin,120.38,111.35,0.00),v40,fine,tPen\WObj:=wPaper;
    MoveL Offs(pOrigin,120.38,111.35,6.00),v60,z5,tPen\WObj:=wPaper;
    MoveL Offs(pOrigin,122.48,112.24,6.00),vTravel,z5,tPen\WObj:=wPaper;
    MoveL Offs(pOrigin,122.48,112.24,0.00),v60,z0,tPen\WObj:=wPaper;
    MoveL Offs(pOrigin,120.97,113.74,0.00),v40,fine,tPen\WObj:=wPaper;
    MoveL Offs(pOrigin,120.97,113.74,6.00),v60,z5,tPen\WObj:=wPaper;
    MoveL Offs(pOrigin,117.40,111.25,6.00),vTravel,z5,tPen\WObj:=wPaper;
    MoveL Offs(pOrigin,117.40,111.25,0.00),v60,z0,tPen\WObj:=wPaper;
    MoveL Offs(pOrigin,117.19,111.46,0.00),v40,z0,tPen\WObj:=wPaper;
    MoveL Offs(pOrigin,116.55,111.25,0.00),v40,z0,tPen\WObj:=wPaper;
    MoveL Offs(pOrigin,116.12,110.40,0.00),v40,fine,tPen\WObj:=wPaper;
    MoveL Offs(pOrigin,116.12,110.40,6.00),v60,z5,tPen\WObj:=wPaper;
    MoveL Offs(pOrigin,110.39,110.04,6.00),vTravel,z5,tPen\WObj:=wPaper;
    MoveL Offs(pOrigin,110.39,110.04,0.00),v60,z0,tPen\WObj:=wPaper;
    MoveL Offs(pOrigin,108.90,110.04,0.00),v40,fine,tPen\WObj:=wPaper;
    MoveL Offs(pOrigin,108.90,110.04,6.00),v60,z5,tPen\WObj:=wPaper;
    MoveL Offs(pOrigin,109.75,108.70,6.00),vTravel,z5,tPen\WObj:=wPaper;
    MoveL Offs(pOrigin,109.75,108.70,0.00),v60,z0,tPen\WObj:=wPaper;
    MoveL Offs(pOrigin,109.96,109.12,0.00),v40,z0,tPen\WObj:=wPaper;
    MoveL Offs(pOrigin,109.75,108.70,0.00),v40,fine,tPen\WObj:=wPaper;
    MoveL Offs(pOrigin,109.75,108.70,6.00),v60,z5,tPen\WObj:=wPaper;
    MoveL Offs(pOrigin,107.62,104.76,6.00),vTravel,z5,tPen\WObj:=wPaper;
    MoveL Offs(pOrigin,107.62,104.76,0.00),v60,z0,tPen\WObj:=wPaper;
    MoveL Offs(pOrigin,106.35,104.76,0.00),v40,z0,tPen\WObj:=wPaper;
    MoveL Offs(pOrigin,105.42,105.40,0.00),v40,z0,tPen\WObj:=wPaper;
    MoveL Offs(pOrigin,109.48,101.34,0.00),v40,z0,tPen\WObj:=wPaper;
    MoveL Offs(pOrigin,108.88,100.45,0.00),v40,z0,tPen\WObj:=wPaper;
    MoveL Offs(pOrigin,104.97,104.35,0.00),v40,z0,tPen\WObj:=wPaper;
    MoveL Offs(pOrigin,104.53,103.31,0.00),v40,z0,tPen\WObj:=wPaper;
    MoveL Offs(pOrigin,108.28,99.55,0.00),v40,fine,tPen\WObj:=wPaper;
    MoveL Offs(pOrigin,108.28,99.55,6.00),v60,z5,tPen\WObj:=wPaper;
    MoveL Offs(pOrigin,111.13,99.69,6.00),vTravel,z5,tPen\WObj:=wPaper;
    MoveL Offs(pOrigin,111.13,99.69,0.00),v60,z0,tPen\WObj:=wPaper;
    MoveL Offs(pOrigin,112.78,98.04,0.00),v40,z0,tPen\WObj:=wPaper;
    MoveL Offs(pOrigin,113.83,98.48,0.00),v40,z0,tPen\WObj:=wPaper;
    MoveL Offs(pOrigin,112.18,100.14,0.00),v40,z0,tPen\WObj:=wPaper;
    MoveL Offs(pOrigin,113.07,100.73,0.00),v40,z0,tPen\WObj:=wPaper;
    MoveL Offs(pOrigin,114.73,99.08,0.00),v40,z0,tPen\WObj:=wPaper;
    MoveL Offs(pOrigin,113.96,99.32,0.00),v40,z0,tPen\WObj:=wPaper;
    MoveL Offs(pOrigin,115.62,100.97,0.00),v40,fine,tPen\WObj:=wPaper;
    MoveL Offs(pOrigin,115.62,100.97,6.00),v60,z5,tPen\WObj:=wPaper;
    MoveL Offs(pOrigin,111.45,98.71,6.00),vTravel,z5,tPen\WObj:=wPaper;
    MoveL Offs(pOrigin,111.45,98.71,0.00),v60,z0,tPen\WObj:=wPaper;
    MoveL Offs(pOrigin,106.14,95.88,0.00),v40,z0,tPen\WObj:=wPaper;
    MoveL Offs(pOrigin,105.07,95.95,0.00),v40,z0,tPen\WObj:=wPaper;
    MoveL Offs(pOrigin,107.34,103.81,0.00),v40,z0,tPen\WObj:=wPaper;
    MoveL Offs(pOrigin,109.25,108.28,0.00),v40,z0,tPen\WObj:=wPaper;
    MoveL Offs(pOrigin,110.60,110.40,0.00),v40,z0,tPen\WObj:=wPaper;
    MoveL Offs(pOrigin,114.85,115.29,0.00),v40,z0,tPen\WObj:=wPaper;
    MoveL Offs(pOrigin,117.26,119.32,0.00),v40,z0,tPen\WObj:=wPaper;
    MoveL Offs(pOrigin,118.25,122.72,0.00),v40,z0,tPen\WObj:=wPaper;
    MoveL Offs(pOrigin,119.31,129.10,0.00),v40,z0,tPen\WObj:=wPaper;
    MoveL Offs(pOrigin,120.59,131.44,0.00),v40,z0,tPen\WObj:=wPaper;
    MoveL Offs(pOrigin,122.07,132.07,0.00),v40,z0,tPen\WObj:=wPaper;
    MoveL Offs(pOrigin,123.78,132.29,0.00),v40,z0,tPen\WObj:=wPaper;
    MoveL Offs(pOrigin,132.70,131.23,0.00),v40,z0,tPen\WObj:=wPaper;
    MoveL Offs(pOrigin,143.96,128.46,0.00),v40,z0,tPen\WObj:=wPaper;
    MoveL Offs(pOrigin,146.09,128.25,0.00),v40,z0,tPen\WObj:=wPaper;
    MoveL Offs(pOrigin,150.76,126.34,0.00),v40,z0,tPen\WObj:=wPaper;
    MoveL Offs(pOrigin,150.15,126.38,0.00),v40,z0,tPen\WObj:=wPaper;
    MoveL Offs(pOrigin,147.89,128.64,0.00),v40,fine,tPen\WObj:=wPaper;
    MoveL Offs(pOrigin,147.89,128.64,6.00),v60,z5,tPen\WObj:=wPaper;
    MoveL Offs(pOrigin,149.54,128.48,6.00),vTravel,z5,tPen\WObj:=wPaper;
    MoveL Offs(pOrigin,149.54,128.48,0.00),v60,z0,tPen\WObj:=wPaper;
    MoveL Offs(pOrigin,144.58,133.44,0.00),v40,fine,tPen\WObj:=wPaper;
    MoveL Offs(pOrigin,144.58,133.44,6.00),v60,z5,tPen\WObj:=wPaper;
    MoveL Offs(pOrigin,146.58,134.92,6.00),vTravel,z5,tPen\WObj:=wPaper;
    MoveL Offs(pOrigin,146.58,134.92,0.00),v60,z0,tPen\WObj:=wPaper;
    MoveL Offs(pOrigin,147.63,135.98,0.00),v40,z0,tPen\WObj:=wPaper;
    MoveL Offs(pOrigin,148.68,135.53,0.00),v40,z0,tPen\WObj:=wPaper;
    MoveL Offs(pOrigin,147.63,134.48,0.00),v40,fine,tPen\WObj:=wPaper;
    MoveL Offs(pOrigin,147.63,134.48,6.00),v60,z5,tPen\WObj:=wPaper;
    MoveL Offs(pOrigin,149.57,133.43,6.00),vTravel,z5,tPen\WObj:=wPaper;
    MoveL Offs(pOrigin,149.57,133.43,0.00),v60,z0,tPen\WObj:=wPaper;
    MoveL Offs(pOrigin,150.92,134.79,0.00),v40,fine,tPen\WObj:=wPaper;
    MoveL Offs(pOrigin,150.92,134.79,6.00),v60,z5,tPen\WObj:=wPaper;
    MoveL Offs(pOrigin,148.96,131.34,6.00),vTravel,z5,tPen\WObj:=wPaper;
    MoveL Offs(pOrigin,148.96,131.34,0.00),v60,z0,tPen\WObj:=wPaper;
    MoveL Offs(pOrigin,148.06,130.43,0.00),v40,fine,tPen\WObj:=wPaper;
    MoveL Offs(pOrigin,148.06,130.43,6.00),v60,z5,tPen\WObj:=wPaper;
    MoveL Offs(pOrigin,140.87,130.71,6.00),vTravel,z5,tPen\WObj:=wPaper;
  ENDPROC

  PROC DrawPart284()
    MoveL Offs(pOrigin,140.87,130.71,0.00),v60,z0,tPen\WObj:=wPaper;
    MoveL Offs(pOrigin,139.52,129.36,0.00),v40,fine,tPen\WObj:=wPaper;
    MoveL Offs(pOrigin,139.52,129.36,6.00),v60,z5,tPen\WObj:=wPaper;
    MoveL Offs(pOrigin,137.43,131.75,6.00),vTravel,z5,tPen\WObj:=wPaper;
    MoveL Offs(pOrigin,137.43,131.75,0.00),v60,z0,tPen\WObj:=wPaper;
    MoveL Offs(pOrigin,135.78,130.10,0.00),v40,fine,tPen\WObj:=wPaper;
    MoveL Offs(pOrigin,135.78,130.10,6.00),v60,z5,tPen\WObj:=wPaper;
    MoveL Offs(pOrigin,133.54,132.34,6.00),vTravel,z5,tPen\WObj:=wPaper;
    MoveL Offs(pOrigin,133.54,132.34,0.00),v60,z0,tPen\WObj:=wPaper;
    MoveL Offs(pOrigin,132.19,130.98,0.00),v40,fine,tPen\WObj:=wPaper;
    MoveL Offs(pOrigin,132.19,130.98,6.00),v60,z5,tPen\WObj:=wPaper;
    MoveL Offs(pOrigin,139.79,133.76,6.00),vTravel,z5,tPen\WObj:=wPaper;
    MoveL Offs(pOrigin,139.79,133.76,0.00),v60,z0,tPen\WObj:=wPaper;
    MoveL Offs(pOrigin,140.99,132.55,0.00),v40,fine,tPen\WObj:=wPaper;
    MoveL Offs(pOrigin,140.99,132.55,6.00),v60,z5,tPen\WObj:=wPaper;
    MoveL Offs(pOrigin,147.41,139.58,6.00),vTravel,z5,tPen\WObj:=wPaper;
    MoveL Offs(pOrigin,147.41,139.58,0.00),v60,z0,tPen\WObj:=wPaper;
    MoveL Offs(pOrigin,142.45,144.53,0.00),v40,fine,tPen\WObj:=wPaper;
    MoveL Offs(pOrigin,142.45,144.53,6.00),v60,z5,tPen\WObj:=wPaper;
    MoveL Offs(pOrigin,146.94,147.80,6.00),vTravel,z5,tPen\WObj:=wPaper;
    MoveL Offs(pOrigin,146.94,147.80,0.00),v60,z0,tPen\WObj:=wPaper;
    MoveL Offs(pOrigin,147.15,147.38,0.00),v40,z0,tPen\WObj:=wPaper;
    MoveL Offs(pOrigin,146.94,147.80,0.00),v40,fine,tPen\WObj:=wPaper;
    MoveL Offs(pOrigin,146.94,147.80,6.00),v60,z5,tPen\WObj:=wPaper;
    MoveL Offs(pOrigin,146.48,152.75,6.00),vTravel,z5,tPen\WObj:=wPaper;
    MoveL Offs(pOrigin,146.48,152.75,0.00),v60,z0,tPen\WObj:=wPaper;
    MoveL Offs(pOrigin,147.38,153.65,0.00),v40,fine,tPen\WObj:=wPaper;
    MoveL Offs(pOrigin,147.38,153.65,6.00),v60,z5,tPen\WObj:=wPaper;
    MoveL Offs(pOrigin,144.81,154.39,6.00),vTravel,z5,tPen\WObj:=wPaper;
    MoveL Offs(pOrigin,144.81,154.39,0.00),v60,z0,tPen\WObj:=wPaper;
    MoveL Offs(pOrigin,145.24,153.96,0.00),v40,z0,tPen\WObj:=wPaper;
    MoveL Offs(pOrigin,144.81,154.39,0.00),v40,fine,tPen\WObj:=wPaper;
    MoveL Offs(pOrigin,144.81,154.39,6.00),v60,z5,tPen\WObj:=wPaper;
    MoveL Offs(pOrigin,143.32,157.57,6.00),vTravel,z5,tPen\WObj:=wPaper;
    MoveL Offs(pOrigin,143.32,157.57,0.00),v60,z0,tPen\WObj:=wPaper;
    MoveL Offs(pOrigin,143.11,158.00,0.00),v40,z0,tPen\WObj:=wPaper;
    MoveL Offs(pOrigin,143.32,157.57,0.00),v40,z0,tPen\WObj:=wPaper;
    MoveL Offs(pOrigin,143.11,157.56,0.00),v40,z0,tPen\WObj:=wPaper;
    MoveL Offs(pOrigin,141.84,157.56,0.00),v40,z0,tPen\WObj:=wPaper;
    MoveL Offs(pOrigin,141.62,157.57,0.00),v40,z0,tPen\WObj:=wPaper;
    MoveL Offs(pOrigin,141.84,157.15,0.00),v40,z0,tPen\WObj:=wPaper;
    MoveL Offs(pOrigin,141.62,157.57,0.00),v40,fine,tPen\WObj:=wPaper;
    MoveL Offs(pOrigin,141.62,157.57,6.00),v60,z5,tPen\WObj:=wPaper;
    MoveL Offs(pOrigin,141.20,159.67,6.00),vTravel,z5,tPen\WObj:=wPaper;
    MoveL Offs(pOrigin,141.20,159.67,0.00),v60,z0,tPen\WObj:=wPaper;
    MoveL Offs(pOrigin,139.93,159.67,0.00),v40,z0,tPen\WObj:=wPaper;
    MoveL Offs(pOrigin,139.93,159.49,0.00),v40,z0,tPen\WObj:=wPaper;
    MoveL Offs(pOrigin,140.14,159.06,0.00),v40,z0,tPen\WObj:=wPaper;
    MoveL Offs(pOrigin,139.93,159.49,0.00),v40,z0,tPen\WObj:=wPaper;
    MoveL Offs(pOrigin,139.50,159.70,0.00),v40,z0,tPen\WObj:=wPaper;
    MoveL Offs(pOrigin,139.29,160.12,0.00),v40,z0,tPen\WObj:=wPaper;
    MoveL Offs(pOrigin,139.50,159.70,0.00),v40,z0,tPen\WObj:=wPaper;
    MoveL Offs(pOrigin,139.02,160.22,0.00),v40,z0,tPen\WObj:=wPaper;
    MoveL Offs(pOrigin,140.37,161.57,0.00),v40,z0,tPen\WObj:=wPaper;
    MoveL Offs(pOrigin,139.93,161.61,0.00),v40,z0,tPen\WObj:=wPaper;
    MoveL Offs(pOrigin,139.71,162.04,0.00),v40,z0,tPen\WObj:=wPaper;
    MoveL Offs(pOrigin,139.93,161.61,0.00),v40,fine,tPen\WObj:=wPaper;
    MoveL Offs(pOrigin,139.93,161.61,6.00),v60,z5,tPen\WObj:=wPaper;
    MoveL Offs(pOrigin,141.20,159.91,6.00),vTravel,z5,tPen\WObj:=wPaper;
    MoveL Offs(pOrigin,141.20,159.91,0.00),v60,z0,tPen\WObj:=wPaper;
    MoveL Offs(pOrigin,140.99,160.34,0.00),v40,z0,tPen\WObj:=wPaper;
    MoveL Offs(pOrigin,141.20,159.91,0.00),v40,fine,tPen\WObj:=wPaper;
    MoveL Offs(pOrigin,141.20,159.91,6.00),v60,z5,tPen\WObj:=wPaper;
    MoveL Offs(pOrigin,139.09,164.32,6.00),vTravel,z5,tPen\WObj:=wPaper;
    MoveL Offs(pOrigin,139.09,164.32,0.00),v60,z0,tPen\WObj:=wPaper;
    MoveL Offs(pOrigin,133.98,169.43,0.00),v40,z0,tPen\WObj:=wPaper;
    MoveL Offs(pOrigin,134.82,169.18,0.00),v40,z0,tPen\WObj:=wPaper;
    MoveL Offs(pOrigin,136.10,169.18,0.00),v40,z0,tPen\WObj:=wPaper;
    MoveL Offs(pOrigin,135.18,168.84,0.00),v40,z0,tPen\WObj:=wPaper;
    MoveL Offs(pOrigin,135.18,166.71,0.00),v40,z0,tPen\WObj:=wPaper;
    MoveL Offs(pOrigin,136.31,167.06,0.00),v40,z0,tPen\WObj:=wPaper;
    MoveL Offs(pOrigin,133.98,167.06,0.00),v40,fine,tPen\WObj:=wPaper;
    MoveL Offs(pOrigin,133.98,167.06,6.00),v60,z5,tPen\WObj:=wPaper;
    MoveL Offs(pOrigin,137.13,169.27,6.00),vTravel,z5,tPen\WObj:=wPaper;
    MoveL Offs(pOrigin,137.13,169.27,0.00),v60,z0,tPen\WObj:=wPaper;
    MoveL Offs(pOrigin,134.73,171.67,0.00),v40,z0,tPen\WObj:=wPaper;
    MoveL Offs(pOrigin,135.17,172.72,0.00),v40,z0,tPen\WObj:=wPaper;
    MoveL Offs(pOrigin,137.58,170.31,0.00),v40,fine,tPen\WObj:=wPaper;
    MoveL Offs(pOrigin,137.58,170.31,6.00),v60,z5,tPen\WObj:=wPaper;
    MoveL Offs(pOrigin,137.16,172.34,6.00),vTravel,z5,tPen\WObj:=wPaper;
    MoveL Offs(pOrigin,137.16,172.34,0.00),v60,z0,tPen\WObj:=wPaper;
    MoveL Offs(pOrigin,136.10,172.34,0.00),v40,z0,tPen\WObj:=wPaper;
    MoveL Offs(pOrigin,136.52,173.40,0.00),v40,z0,tPen\WObj:=wPaper;
    MoveL Offs(pOrigin,137.59,173.40,0.00),v40,z0,tPen\WObj:=wPaper;
    MoveL Offs(pOrigin,137.80,174.46,0.00),v40,z0,tPen\WObj:=wPaper;
    MoveL Offs(pOrigin,136.74,174.46,0.00),v40,z0,tPen\WObj:=wPaper;
    MoveL Offs(pOrigin,136.95,175.51,0.00),v40,z0,tPen\WObj:=wPaper;
    MoveL Offs(pOrigin,138.01,175.51,0.00),v40,fine,tPen\WObj:=wPaper;
    MoveL Offs(pOrigin,138.01,175.51,6.00),v60,z5,tPen\WObj:=wPaper;
    MoveL Offs(pOrigin,138.62,173.76,6.00),vTravel,z5,tPen\WObj:=wPaper;
    MoveL Offs(pOrigin,138.62,173.76,0.00),v60,z0,tPen\WObj:=wPaper;
    MoveL Offs(pOrigin,136.06,176.31,0.00),v40,fine,tPen\WObj:=wPaper;
    MoveL Offs(pOrigin,136.06,176.31,6.00),v60,z5,tPen\WObj:=wPaper;
    MoveL Offs(pOrigin,142.97,169.40,6.00),vTravel,z5,tPen\WObj:=wPaper;
    MoveL Offs(pOrigin,142.97,169.40,0.00),v60,z0,tPen\WObj:=wPaper;
    MoveL Offs(pOrigin,151.39,160.98,0.00),v40,fine,tPen\WObj:=wPaper;
    MoveL Offs(pOrigin,151.39,160.98,6.00),v60,z5,tPen\WObj:=wPaper;
    MoveL Offs(pOrigin,150.76,159.67,6.00),vTravel,z5,tPen\WObj:=wPaper;
    MoveL Offs(pOrigin,150.76,159.67,0.00),v60,z0,tPen\WObj:=wPaper;
    MoveL Offs(pOrigin,149.06,159.67,0.00),v40,z0,tPen\WObj:=wPaper;
    MoveL Offs(pOrigin,149.97,160.12,0.00),v40,z0,tPen\WObj:=wPaper;
    MoveL Offs(pOrigin,149.97,158.21,0.00),v40,fine,tPen\WObj:=wPaper;
    MoveL Offs(pOrigin,149.97,158.21,6.00),v60,z5,tPen\WObj:=wPaper;
    MoveL Offs(pOrigin,152.29,158.58,6.00),vTravel,z5,tPen\WObj:=wPaper;
    MoveL Offs(pOrigin,152.29,158.58,0.00),v60,z0,tPen\WObj:=wPaper;
    MoveL Offs(pOrigin,143.88,167.00,0.00),v40,fine,tPen\WObj:=wPaper;
    MoveL Offs(pOrigin,143.88,167.00,6.00),v60,z5,tPen\WObj:=wPaper;
    MoveL Offs(pOrigin,145.88,165.23,6.00),vTravel,z5,tPen\WObj:=wPaper;
    MoveL Offs(pOrigin,145.88,165.23,0.00),v60,z0,tPen\WObj:=wPaper;
    MoveL Offs(pOrigin,145.66,165.65,0.00),v40,z0,tPen\WObj:=wPaper;
    MoveL Offs(pOrigin,145.88,165.23,0.00),v40,fine,tPen\WObj:=wPaper;
    MoveL Offs(pOrigin,145.88,165.23,6.00),v60,z5,tPen\WObj:=wPaper;
    MoveL Offs(pOrigin,145.39,164.00,6.00),vTravel,z5,tPen\WObj:=wPaper;
    MoveL Offs(pOrigin,145.39,164.00,0.00),v60,z0,tPen\WObj:=wPaper;
    MoveL Offs(pOrigin,152.90,156.49,0.00),v40,fine,tPen\WObj:=wPaper;
    MoveL Offs(pOrigin,152.90,156.49,6.00),v60,z5,tPen\WObj:=wPaper;
    MoveL Offs(pOrigin,153.81,154.09,6.00),vTravel,z5,tPen\WObj:=wPaper;
    MoveL Offs(pOrigin,153.81,154.09,0.00),v60,z0,tPen\WObj:=wPaper;
    MoveL Offs(pOrigin,146.59,161.30,0.00),v40,fine,tPen\WObj:=wPaper;
    MoveL Offs(pOrigin,146.59,161.30,6.00),v60,z5,tPen\WObj:=wPaper;
  ENDPROC

  PROC DrawPart285()
    MoveL Offs(pOrigin,146.97,166.68,6.00),vTravel,z5,tPen\WObj:=wPaper;
    MoveL Offs(pOrigin,146.97,166.68,0.00),v60,z0,tPen\WObj:=wPaper;
    MoveL Offs(pOrigin,148.63,168.34,0.00),v40,fine,tPen\WObj:=wPaper;
    MoveL Offs(pOrigin,148.63,168.34,6.00),v60,z5,tPen\WObj:=wPaper;
    MoveL Offs(pOrigin,150.06,154.85,6.00),vTravel,z5,tPen\WObj:=wPaper;
    MoveL Offs(pOrigin,150.06,154.85,0.00),v60,z0,tPen\WObj:=wPaper;
    MoveL Offs(pOrigin,155.02,149.89,0.00),v40,fine,tPen\WObj:=wPaper;
    MoveL Offs(pOrigin,155.02,149.89,6.00),v60,z5,tPen\WObj:=wPaper;
    MoveL Offs(pOrigin,154.38,148.06,6.00),vTravel,z5,tPen\WObj:=wPaper;
    MoveL Offs(pOrigin,154.38,148.06,0.00),v60,z0,tPen\WObj:=wPaper;
    MoveL Offs(pOrigin,153.31,148.06,0.00),v40,z0,tPen\WObj:=wPaper;
    MoveL Offs(pOrigin,152.18,148.25,0.00),v40,z0,tPen\WObj:=wPaper;
    MoveL Offs(pOrigin,157.13,143.29,0.00),v40,fine,tPen\WObj:=wPaper;
    MoveL Offs(pOrigin,157.13,143.29,6.00),v60,z5,tPen\WObj:=wPaper;
    MoveL Offs(pOrigin,152.46,141.64,6.00),vTravel,z5,tPen\WObj:=wPaper;
    MoveL Offs(pOrigin,152.46,141.64,0.00),v60,z0,tPen\WObj:=wPaper;
    MoveL Offs(pOrigin,152.25,142.06,0.00),v40,z0,tPen\WObj:=wPaper;
    MoveL Offs(pOrigin,152.46,141.64,0.00),v40,fine,tPen\WObj:=wPaper;
    MoveL Offs(pOrigin,152.46,141.64,6.00),v60,z5,tPen\WObj:=wPaper;
    MoveL Offs(pOrigin,158.20,125.28,6.00),vTravel,z5,tPen\WObj:=wPaper;
    MoveL Offs(pOrigin,158.20,125.28,0.00),v60,z0,tPen\WObj:=wPaper;
    MoveL Offs(pOrigin,157.56,125.91,0.00),v40,z0,tPen\WObj:=wPaper;
    MoveL Offs(pOrigin,158.20,125.28,0.00),v40,z0,tPen\WObj:=wPaper;
    MoveL Offs(pOrigin,157.77,124.21,0.00),v40,z0,tPen\WObj:=wPaper;
    MoveL Offs(pOrigin,157.99,123.79,0.00),v40,z0,tPen\WObj:=wPaper;
    MoveL Offs(pOrigin,157.77,124.21,0.00),v40,z0,tPen\WObj:=wPaper;
    MoveL Offs(pOrigin,158.41,123.57,0.00),v40,z0,tPen\WObj:=wPaper;
    MoveL Offs(pOrigin,158.62,123.15,0.00),v40,z0,tPen\WObj:=wPaper;
    MoveL Offs(pOrigin,158.41,123.57,0.00),v40,fine,tPen\WObj:=wPaper;
    MoveL Offs(pOrigin,158.41,123.57,6.00),v60,z5,tPen\WObj:=wPaper;
    MoveL Offs(pOrigin,155.71,120.82,6.00),vTravel,z5,tPen\WObj:=wPaper;
    MoveL Offs(pOrigin,155.71,120.82,0.00),v60,z0,tPen\WObj:=wPaper;
    MoveL Offs(pOrigin,157.51,119.02,0.00),v40,fine,tPen\WObj:=wPaper;
    MoveL Offs(pOrigin,157.51,119.02,6.00),v60,z5,tPen\WObj:=wPaper;
    MoveL Offs(pOrigin,160.11,116.38,6.00),vTravel,z5,tPen\WObj:=wPaper;
    MoveL Offs(pOrigin,160.11,116.38,0.00),v60,z0,tPen\WObj:=wPaper;
    MoveL Offs(pOrigin,161.81,116.38,0.00),v40,fine,tPen\WObj:=wPaper;
    MoveL Offs(pOrigin,161.81,116.38,6.00),v60,z5,tPen\WObj:=wPaper;
    MoveL Offs(pOrigin,160.53,115.92,6.00),vTravel,z5,tPen\WObj:=wPaper;
    MoveL Offs(pOrigin,160.53,115.92,0.00),v60,z0,tPen\WObj:=wPaper;
    MoveL Offs(pOrigin,160.53,113.59,0.00),v40,fine,tPen\WObj:=wPaper;
    MoveL Offs(pOrigin,160.53,113.59,6.00),v60,z5,tPen\WObj:=wPaper;
    MoveL Offs(pOrigin,154.70,105.40,6.00),vTravel,z5,tPen\WObj:=wPaper;
    MoveL Offs(pOrigin,154.70,105.40,0.00),v60,z0,tPen\WObj:=wPaper;
    MoveL Offs(pOrigin,151.40,108.70,0.00),v40,fine,tPen\WObj:=wPaper;
    MoveL Offs(pOrigin,151.40,108.70,6.00),v60,z5,tPen\WObj:=wPaper;
    MoveL Offs(pOrigin,152.62,100.01,6.00),vTravel,z5,tPen\WObj:=wPaper;
    MoveL Offs(pOrigin,152.62,100.01,0.00),v60,z0,tPen\WObj:=wPaper;
    MoveL Offs(pOrigin,155.03,97.61,0.00),v40,fine,tPen\WObj:=wPaper;
    MoveL Offs(pOrigin,155.03,97.61,6.00),v60,z5,tPen\WObj:=wPaper;
    MoveL Offs(pOrigin,152.03,97.62,6.00),vTravel,z5,tPen\WObj:=wPaper;
    MoveL Offs(pOrigin,152.03,97.62,0.00),v60,z0,tPen\WObj:=wPaper;
    MoveL Offs(pOrigin,149.63,100.02,0.00),v40,fine,tPen\WObj:=wPaper;
    MoveL Offs(pOrigin,149.63,100.02,6.00),v60,z5,tPen\WObj:=wPaper;
    MoveL Offs(pOrigin,146.05,93.14,6.00),vTravel,z5,tPen\WObj:=wPaper;
    MoveL Offs(pOrigin,146.05,93.14,0.00),v60,z0,tPen\WObj:=wPaper;
    MoveL Offs(pOrigin,156.87,82.32,0.00),v40,fine,tPen\WObj:=wPaper;
    MoveL Offs(pOrigin,156.87,82.32,6.00),v60,z5,tPen\WObj:=wPaper;
    MoveL Offs(pOrigin,159.26,80.47,6.00),vTravel,z5,tPen\WObj:=wPaper;
    MoveL Offs(pOrigin,159.26,80.47,0.00),v60,z0,tPen\WObj:=wPaper;
    MoveL Offs(pOrigin,160.54,80.47,0.00),v40,fine,tPen\WObj:=wPaper;
    MoveL Offs(pOrigin,160.54,80.47,6.00),v60,z5,tPen\WObj:=wPaper;
    MoveL Offs(pOrigin,165.85,86.79,6.00),vTravel,z5,tPen\WObj:=wPaper;
    MoveL Offs(pOrigin,165.85,86.79,0.00),v60,z0,tPen\WObj:=wPaper;
    MoveL Offs(pOrigin,159.23,93.40,0.00),v40,z0,tPen\WObj:=wPaper;
    MoveL Offs(pOrigin,159.83,94.30,0.00),v40,z0,tPen\WObj:=wPaper;
    MoveL Offs(pOrigin,165.39,88.74,0.00),v40,fine,tPen\WObj:=wPaper;
    MoveL Offs(pOrigin,165.39,88.74,6.00),v60,z5,tPen\WObj:=wPaper;
    MoveL Offs(pOrigin,166.82,90.94,6.00),vTravel,z5,tPen\WObj:=wPaper;
    MoveL Offs(pOrigin,166.82,90.94,0.00),v60,z0,tPen\WObj:=wPaper;
    MoveL Offs(pOrigin,169.37,93.50,0.00),v40,fine,tPen\WObj:=wPaper;
    MoveL Offs(pOrigin,169.37,93.50,6.00),v60,z5,tPen\WObj:=wPaper;
    MoveL Offs(pOrigin,167.98,94.46,6.00),vTravel,z5,tPen\WObj:=wPaper;
    MoveL Offs(pOrigin,167.98,94.46,0.00),v60,z0,tPen\WObj:=wPaper;
    MoveL Offs(pOrigin,167.12,94.53,0.00),v40,z0,tPen\WObj:=wPaper;
    MoveL Offs(pOrigin,166.77,94.89,0.00),v40,z0,tPen\WObj:=wPaper;
    MoveL Offs(pOrigin,167.12,95.95,0.00),v40,z0,tPen\WObj:=wPaper;
    MoveL Offs(pOrigin,168.40,96.38,0.00),v40,z0,tPen\WObj:=wPaper;
    MoveL Offs(pOrigin,168.82,95.53,0.00),v40,fine,tPen\WObj:=wPaper;
    MoveL Offs(pOrigin,168.82,95.53,6.00),v60,z5,tPen\WObj:=wPaper;
    MoveL Offs(pOrigin,166.91,95.26,6.00),vTravel,z5,tPen\WObj:=wPaper;
    MoveL Offs(pOrigin,166.91,95.26,0.00),v60,z0,tPen\WObj:=wPaper;
    MoveL Offs(pOrigin,161.81,95.26,0.00),v40,z0,tPen\WObj:=wPaper;
    MoveL Offs(pOrigin,161.58,94.25,0.00),v40,z0,tPen\WObj:=wPaper;
    MoveL Offs(pOrigin,161.58,90.64,0.00),v40,z0,tPen\WObj:=wPaper;
    MoveL Offs(pOrigin,162.24,91.49,0.00),v40,z0,tPen\WObj:=wPaper;
    MoveL Offs(pOrigin,161.39,82.99,0.00),v40,z0,tPen\WObj:=wPaper;
    MoveL Offs(pOrigin,159.83,77.68,0.00),v40,z0,tPen\WObj:=wPaper;
    MoveL Offs(pOrigin,160.11,77.32,0.00),v40,z0,tPen\WObj:=wPaper;
    MoveL Offs(pOrigin,167.76,74.70,0.00),v40,z0,tPen\WObj:=wPaper;
    MoveL Offs(pOrigin,167.98,75.55,0.00),v40,z0,tPen\WObj:=wPaper;
    MoveL Offs(pOrigin,165.21,82.14,0.00),v40,z0,tPen\WObj:=wPaper;
    MoveL Offs(pOrigin,162.88,90.85,0.00),v40,z0,tPen\WObj:=wPaper;
    MoveL Offs(pOrigin,162.31,91.70,0.00),v40,z0,tPen\WObj:=wPaper;
    MoveL Offs(pOrigin,162.45,92.12,0.00),v40,fine,tPen\WObj:=wPaper;
    MoveL Offs(pOrigin,162.45,92.12,6.00),v60,z5,tPen\WObj:=wPaper;
    MoveL Offs(pOrigin,160.54,93.61,6.00),vTravel,z5,tPen\WObj:=wPaper;
    MoveL Offs(pOrigin,160.54,93.61,0.00),v60,z0,tPen\WObj:=wPaper;
    MoveL Offs(pOrigin,160.75,94.04,0.00),v40,z0,tPen\WObj:=wPaper;
    MoveL Offs(pOrigin,160.54,93.61,0.00),v40,fine,tPen\WObj:=wPaper;
    MoveL Offs(pOrigin,160.54,93.61,6.00),v60,z5,tPen\WObj:=wPaper;
    MoveL Offs(pOrigin,159.77,89.87,6.00),vTravel,z5,tPen\WObj:=wPaper;
    MoveL Offs(pOrigin,159.77,89.87,0.00),v60,z0,tPen\WObj:=wPaper;
    MoveL Offs(pOrigin,168.04,98.14,0.00),v40,z0,tPen\WObj:=wPaper;
    MoveL Offs(pOrigin,167.46,98.62,0.00),v40,z0,tPen\WObj:=wPaper;
    MoveL Offs(pOrigin,194.65,71.42,0.00),v40,z0,tPen\WObj:=wPaper;
    MoveL Offs(pOrigin,194.47,72.30,0.00),v40,z0,tPen\WObj:=wPaper;
    MoveL Offs(pOrigin,198.68,76.51,0.00),v40,fine,tPen\WObj:=wPaper;
    MoveL Offs(pOrigin,198.68,76.51,6.00),v60,z5,tPen\WObj:=wPaper;
    MoveL Offs(pOrigin,179.90,95.13,6.00),vTravel,z5,tPen\WObj:=wPaper;
    MoveL Offs(pOrigin,179.90,95.13,0.00),v60,z0,tPen\WObj:=wPaper;
    MoveL Offs(pOrigin,179.15,95.89,0.00),v40,z0,tPen\WObj:=wPaper;
    MoveL Offs(pOrigin,179.60,96.93,0.00),v40,z0,tPen\WObj:=wPaper;
    MoveL Offs(pOrigin,180.50,96.03,0.00),v40,z0,tPen\WObj:=wPaper;
    MoveL Offs(pOrigin,181.09,96.93,0.00),v40,z0,tPen\WObj:=wPaper;
    MoveL Offs(pOrigin,180.04,97.98,0.00),v40,z0,tPen\WObj:=wPaper;
    MoveL Offs(pOrigin,180.49,99.03,0.00),v40,z0,tPen\WObj:=wPaper;
    MoveL Offs(pOrigin,181.69,97.83,0.00),v40,z0,tPen\WObj:=wPaper;
    MoveL Offs(pOrigin,182.14,98.87,0.00),v40,z0,tPen\WObj:=wPaper;
    MoveL Offs(pOrigin,181.09,99.92,0.00),v40,z0,tPen\WObj:=wPaper;
  ENDPROC

  PROC DrawPart286()
    MoveL Offs(pOrigin,181.53,100.97,0.00),v40,z0,tPen\WObj:=wPaper;
    MoveL Offs(pOrigin,182.73,99.77,0.00),v40,z0,tPen\WObj:=wPaper;
    MoveL Offs(pOrigin,183.48,100.52,0.00),v40,z0,tPen\WObj:=wPaper;
    MoveL Offs(pOrigin,182.13,101.87,0.00),v40,z0,tPen\WObj:=wPaper;
    MoveL Offs(pOrigin,182.57,102.92,0.00),v40,z0,tPen\WObj:=wPaper;
    MoveL Offs(pOrigin,184.08,101.41,0.00),v40,z0,tPen\WObj:=wPaper;
    MoveL Offs(pOrigin,184.52,102.46,0.00),v40,z0,tPen\WObj:=wPaper;
    MoveL Offs(pOrigin,183.17,103.81,0.00),v40,z0,tPen\WObj:=wPaper;
    MoveL Offs(pOrigin,183.93,103.58,0.00),v40,z0,tPen\WObj:=wPaper;
    MoveL Offs(pOrigin,185.73,105.38,0.00),v40,fine,tPen\WObj:=wPaper;
    MoveL Offs(pOrigin,185.73,105.38,6.00),v60,z5,tPen\WObj:=wPaper;
    MoveL Offs(pOrigin,184.76,108.28,6.00),vTravel,z5,tPen\WObj:=wPaper;
    MoveL Offs(pOrigin,184.76,108.28,0.00),v60,z0,tPen\WObj:=wPaper;
    MoveL Offs(pOrigin,186.25,109.76,0.00),v40,z0,tPen\WObj:=wPaper;
    MoveL Offs(pOrigin,184.76,108.28,0.00),v40,fine,tPen\WObj:=wPaper;
    MoveL Offs(pOrigin,184.76,108.28,6.00),v60,z5,tPen\WObj:=wPaper;
    MoveL Offs(pOrigin,187.24,108.38,6.00),vTravel,z5,tPen\WObj:=wPaper;
    MoveL Offs(pOrigin,187.24,108.38,0.00),v60,z0,tPen\WObj:=wPaper;
    MoveL Offs(pOrigin,191.45,112.59,0.00),v40,z0,tPen\WObj:=wPaper;
    MoveL Offs(pOrigin,191.99,112.74,0.00),v40,z0,tPen\WObj:=wPaper;
    MoveL Offs(pOrigin,192.84,113.59,0.00),v40,z0,tPen\WObj:=wPaper;
    MoveL Offs(pOrigin,191.99,112.74,0.00),v40,fine,tPen\WObj:=wPaper;
    MoveL Offs(pOrigin,191.99,112.74,6.00),v60,z5,tPen\WObj:=wPaper;
    MoveL Offs(pOrigin,190.50,111.25,6.00),vTravel,z5,tPen\WObj:=wPaper;
    MoveL Offs(pOrigin,190.50,111.25,0.00),v60,z0,tPen\WObj:=wPaper;
    MoveL Offs(pOrigin,191.35,112.10,0.00),v40,z0,tPen\WObj:=wPaper;
    MoveL Offs(pOrigin,190.50,111.25,0.00),v40,fine,tPen\WObj:=wPaper;
    MoveL Offs(pOrigin,190.50,111.25,6.00),v60,z5,tPen\WObj:=wPaper;
    MoveL Offs(pOrigin,188.16,108.70,6.00),vTravel,z5,tPen\WObj:=wPaper;
    MoveL Offs(pOrigin,188.16,108.70,0.00),v60,z0,tPen\WObj:=wPaper;
    MoveL Offs(pOrigin,188.59,109.12,0.00),v40,z0,tPen\WObj:=wPaper;
    MoveL Offs(pOrigin,188.16,108.70,0.00),v40,fine,tPen\WObj:=wPaper;
    MoveL Offs(pOrigin,188.16,108.70,6.00),v60,z5,tPen\WObj:=wPaper;
    MoveL Offs(pOrigin,179.43,101.58,6.00),vTravel,z5,tPen\WObj:=wPaper;
    MoveL Offs(pOrigin,179.43,101.58,0.00),v60,z0,tPen\WObj:=wPaper;
    MoveL Offs(pOrigin,178.08,102.93,0.00),v40,z0,tPen\WObj:=wPaper;
    MoveL Offs(pOrigin,177.18,102.33,0.00),v40,z0,tPen\WObj:=wPaper;
    MoveL Offs(pOrigin,178.69,100.83,0.00),v40,z0,tPen\WObj:=wPaper;
    MoveL Offs(pOrigin,177.94,100.08,0.00),v40,z0,tPen\WObj:=wPaper;
    MoveL Offs(pOrigin,176.59,101.44,0.00),v40,z0,tPen\WObj:=wPaper;
    MoveL Offs(pOrigin,175.69,100.84,0.00),v40,z0,tPen\WObj:=wPaper;
    MoveL Offs(pOrigin,177.34,99.19,0.00),v40,z0,tPen\WObj:=wPaper;
    MoveL Offs(pOrigin,176.90,100.20,0.00),v40,z0,tPen\WObj:=wPaper;
    MoveL Offs(pOrigin,177.54,100.84,0.00),v40,z0,tPen\WObj:=wPaper;
    MoveL Offs(pOrigin,176.90,100.20,0.00),v40,fine,tPen\WObj:=wPaper;
    MoveL Offs(pOrigin,176.90,100.20,6.00),v60,z5,tPen\WObj:=wPaper;
    MoveL Offs(pOrigin,174.35,97.65,6.00),vTravel,z5,tPen\WObj:=wPaper;
    MoveL Offs(pOrigin,174.35,97.65,0.00),v60,z0,tPen\WObj:=wPaper;
    MoveL Offs(pOrigin,175.20,98.50,0.00),v40,z0,tPen\WObj:=wPaper;
    MoveL Offs(pOrigin,174.35,97.65,0.00),v40,fine,tPen\WObj:=wPaper;
    MoveL Offs(pOrigin,174.35,97.65,6.00),v60,z5,tPen\WObj:=wPaper;
    MoveL Offs(pOrigin,171.78,97.40,6.00),vTravel,z5,tPen\WObj:=wPaper;
    MoveL Offs(pOrigin,171.78,97.40,0.00),v60,z0,tPen\WObj:=wPaper;
    MoveL Offs(pOrigin,166.07,91.69,0.00),v40,z0,tPen\WObj:=wPaper;
    MoveL Offs(pOrigin,166.28,92.09,0.00),v40,z0,tPen\WObj:=wPaper;
    MoveL Offs(pOrigin,168.40,92.09,0.00),v40,fine,tPen\WObj:=wPaper;
    MoveL Offs(pOrigin,168.40,92.09,6.00),v60,z5,tPen\WObj:=wPaper;
    MoveL Offs(pOrigin,169.25,91.03,6.00),vTravel,z5,tPen\WObj:=wPaper;
    MoveL Offs(pOrigin,169.25,91.03,0.00),v60,z0,tPen\WObj:=wPaper;
    MoveL Offs(pOrigin,167.34,91.03,0.00),v40,z0,tPen\WObj:=wPaper;
    MoveL Offs(pOrigin,166.70,91.49,0.00),v40,z0,tPen\WObj:=wPaper;
    MoveL Offs(pOrigin,166.27,91.91,0.00),v40,z0,tPen\WObj:=wPaper;
    MoveL Offs(pOrigin,166.70,91.49,0.00),v40,fine,tPen\WObj:=wPaper;
    MoveL Offs(pOrigin,166.70,91.49,6.00),v60,z5,tPen\WObj:=wPaper;
    MoveL Offs(pOrigin,165.81,93.61,6.00),vTravel,z5,tPen\WObj:=wPaper;
    MoveL Offs(pOrigin,165.81,93.61,0.00),v60,z0,tPen\WObj:=wPaper;
    MoveL Offs(pOrigin,165.81,96.16,0.00),v40,fine,tPen\WObj:=wPaper;
    MoveL Offs(pOrigin,165.81,96.16,6.00),v60,z5,tPen\WObj:=wPaper;
    MoveL Offs(pOrigin,166.91,97.37,6.00),vTravel,z5,tPen\WObj:=wPaper;
    MoveL Offs(pOrigin,166.91,97.37,0.00),v60,z0,tPen\WObj:=wPaper;
    MoveL Offs(pOrigin,169.46,97.37,0.00),v40,fine,tPen\WObj:=wPaper;
    MoveL Offs(pOrigin,169.46,97.37,6.00),v60,z5,tPen\WObj:=wPaper;
    MoveL Offs(pOrigin,167.34,94.20,6.00),vTravel,z5,tPen\WObj:=wPaper;
    MoveL Offs(pOrigin,167.34,94.20,0.00),v60,z0,tPen\WObj:=wPaper;
    MoveL Offs(pOrigin,165.00,94.20,0.00),v40,fine,tPen\WObj:=wPaper;
    MoveL Offs(pOrigin,165.00,94.20,6.00),v60,z5,tPen\WObj:=wPaper;
    MoveL Offs(pOrigin,168.01,89.15,6.00),vTravel,z5,tPen\WObj:=wPaper;
    MoveL Offs(pOrigin,168.01,89.15,0.00),v60,z0,tPen\WObj:=wPaper;
    MoveL Offs(pOrigin,171.16,92.31,0.00),v40,z0,tPen\WObj:=wPaper;
    MoveL Offs(pOrigin,171.76,91.41,0.00),v40,z0,tPen\WObj:=wPaper;
    MoveL Offs(pOrigin,168.91,88.55,0.00),v40,z0,tPen\WObj:=wPaper;
    MoveL Offs(pOrigin,169.04,88.92,0.00),v40,z0,tPen\WObj:=wPaper;
    MoveL Offs(pOrigin,171.38,88.92,0.00),v40,fine,tPen\WObj:=wPaper;
    MoveL Offs(pOrigin,171.38,88.92,6.00),v60,z5,tPen\WObj:=wPaper;
    MoveL Offs(pOrigin,172.44,87.86,6.00),vTravel,z5,tPen\WObj:=wPaper;
    MoveL Offs(pOrigin,172.44,87.86,0.00),v60,z0,tPen\WObj:=wPaper;
    MoveL Offs(pOrigin,170.31,87.86,0.00),v40,z0,tPen\WObj:=wPaper;
    MoveL Offs(pOrigin,170.31,87.45,0.00),v40,z0,tPen\WObj:=wPaper;
    MoveL Offs(pOrigin,169.68,88.09,0.00),v40,z0,tPen\WObj:=wPaper;
    MoveL Offs(pOrigin,170.31,87.45,0.00),v40,z0,tPen\WObj:=wPaper;
    MoveL Offs(pOrigin,170.40,87.06,0.00),v40,z0,tPen\WObj:=wPaper;
    MoveL Offs(pOrigin,173.25,89.92,0.00),v40,z0,tPen\WObj:=wPaper;
    MoveL Offs(pOrigin,172.51,90.66,0.00),v40,z0,tPen\WObj:=wPaper;
    MoveL Offs(pOrigin,169.65,87.81,0.00),v40,z0,tPen\WObj:=wPaper;
    MoveL Offs(pOrigin,169.46,88.30,0.00),v40,z0,tPen\WObj:=wPaper;
    MoveL Offs(pOrigin,167.98,89.79,0.00),v40,z0,tPen\WObj:=wPaper;
    MoveL Offs(pOrigin,169.46,88.30,0.00),v40,fine,tPen\WObj:=wPaper;
    MoveL Offs(pOrigin,169.46,88.30,6.00),v60,z5,tPen\WObj:=wPaper;
    MoveL Offs(pOrigin,173.93,87.66,6.00),vTravel,z5,tPen\WObj:=wPaper;
    MoveL Offs(pOrigin,173.93,87.66,0.00),v60,z0,tPen\WObj:=wPaper;
    MoveL Offs(pOrigin,172.86,88.72,0.00),v40,z0,tPen\WObj:=wPaper;
    MoveL Offs(pOrigin,173.93,87.66,0.00),v40,fine,tPen\WObj:=wPaper;
    MoveL Offs(pOrigin,173.93,87.66,6.00),v60,z5,tPen\WObj:=wPaper;
    MoveL Offs(pOrigin,160.42,98.19,6.00),vTravel,z5,tPen\WObj:=wPaper;
    MoveL Offs(pOrigin,160.42,98.19,0.00),v60,z0,tPen\WObj:=wPaper;
    MoveL Offs(pOrigin,158.47,100.14,0.00),v40,fine,tPen\WObj:=wPaper;
    MoveL Offs(pOrigin,158.47,100.14,6.00),v60,z5,tPen\WObj:=wPaper;
    MoveL Offs(pOrigin,146.00,92.53,6.00),vTravel,z5,tPen\WObj:=wPaper;
    MoveL Offs(pOrigin,146.00,92.53,0.00),v60,z0,tPen\WObj:=wPaper;
    MoveL Offs(pOrigin,145.10,91.63,0.00),v40,z0,tPen\WObj:=wPaper;
    MoveL Offs(pOrigin,146.09,91.70,0.00),v40,z0,tPen\WObj:=wPaper;
    MoveL Offs(pOrigin,143.11,93.47,0.00),v40,z0,tPen\WObj:=wPaper;
    MoveL Offs(pOrigin,138.86,95.10,0.00),v40,z0,tPen\WObj:=wPaper;
    MoveL Offs(pOrigin,135.46,95.95,0.00),v40,z0,tPen\WObj:=wPaper;
    MoveL Offs(pOrigin,131.43,96.38,0.00),v40,fine,tPen\WObj:=wPaper;
    MoveL Offs(pOrigin,131.43,96.38,6.00),v60,z5,tPen\WObj:=wPaper;
    MoveL Offs(pOrigin,133.76,96.47,6.00),vTravel,z5,tPen\WObj:=wPaper;
    MoveL Offs(pOrigin,133.76,96.47,0.00),v60,z0,tPen\WObj:=wPaper;
    MoveL Offs(pOrigin,135.26,94.97,0.00),v40,fine,tPen\WObj:=wPaper;
    MoveL Offs(pOrigin,135.26,94.97,6.00),v60,z5,tPen\WObj:=wPaper;
  ENDPROC

  PROC DrawPart287()
    MoveL Offs(pOrigin,135.26,96.47,6.00),vTravel,z5,tPen\WObj:=wPaper;
    MoveL Offs(pOrigin,135.26,96.47,0.00),v60,z0,tPen\WObj:=wPaper;
    MoveL Offs(pOrigin,137.36,94.37,0.00),v40,fine,tPen\WObj:=wPaper;
    MoveL Offs(pOrigin,137.36,94.37,6.00),v60,z5,tPen\WObj:=wPaper;
    MoveL Offs(pOrigin,134.76,90.25,6.00),vTravel,z5,tPen\WObj:=wPaper;
    MoveL Offs(pOrigin,134.76,90.25,0.00),v60,z0,tPen\WObj:=wPaper;
    MoveL Offs(pOrigin,132.95,88.44,0.00),v40,z0,tPen\WObj:=wPaper;
    MoveL Offs(pOrigin,132.91,88.92,0.00),v40,z0,tPen\WObj:=wPaper;
    MoveL Offs(pOrigin,136.31,88.92,0.00),v40,z0,tPen\WObj:=wPaper;
    MoveL Offs(pOrigin,136.70,89.20,0.00),v40,z0,tPen\WObj:=wPaper;
    MoveL Offs(pOrigin,134.45,86.95,0.00),v40,z0,tPen\WObj:=wPaper;
    MoveL Offs(pOrigin,135.18,87.66,0.00),v40,z0,tPen\WObj:=wPaper;
    MoveL Offs(pOrigin,135.18,88.94,0.00),v40,fine,tPen\WObj:=wPaper;
    MoveL Offs(pOrigin,135.18,88.94,6.00),v60,z5,tPen\WObj:=wPaper;
    MoveL Offs(pOrigin,136.24,88.30,6.00),vTravel,z5,tPen\WObj:=wPaper;
    MoveL Offs(pOrigin,136.24,88.30,0.00),v60,z0,tPen\WObj:=wPaper;
    MoveL Offs(pOrigin,136.24,87.24,0.00),v40,fine,tPen\WObj:=wPaper;
    MoveL Offs(pOrigin,136.24,87.24,6.00),v60,z5,tPen\WObj:=wPaper;
    MoveL Offs(pOrigin,138.35,87.02,6.00),vTravel,z5,tPen\WObj:=wPaper;
    MoveL Offs(pOrigin,138.35,87.02,0.00),v60,z0,tPen\WObj:=wPaper;
    MoveL Offs(pOrigin,138.35,85.96,0.00),v40,fine,tPen\WObj:=wPaper;
    MoveL Offs(pOrigin,138.35,85.96,6.00),v60,z5,tPen\WObj:=wPaper;
    MoveL Offs(pOrigin,137.14,85.16,6.00),vTravel,z5,tPen\WObj:=wPaper;
    MoveL Offs(pOrigin,137.14,85.16,0.00),v60,z0,tPen\WObj:=wPaper;
    MoveL Offs(pOrigin,139.54,87.57,0.00),v40,z0,tPen\WObj:=wPaper;
    MoveL Offs(pOrigin,140.29,86.82,0.00),v40,z0,tPen\WObj:=wPaper;
    MoveL Offs(pOrigin,136.08,82.61,0.00),v40,fine,tPen\WObj:=wPaper;
    MoveL Offs(pOrigin,136.08,82.61,6.00),v60,z5,tPen\WObj:=wPaper;
    MoveL Offs(pOrigin,134.70,82.09,6.00),vTravel,z5,tPen\WObj:=wPaper;
    MoveL Offs(pOrigin,134.70,82.09,0.00),v60,z0,tPen\WObj:=wPaper;
    MoveL Offs(pOrigin,131.85,84.95,0.00),v40,z0,tPen\WObj:=wPaper;
    MoveL Offs(pOrigin,132.04,84.55,0.00),v40,z0,tPen\WObj:=wPaper;
    MoveL Offs(pOrigin,129.64,82.14,0.00),v40,z0,tPen\WObj:=wPaper;
    MoveL Offs(pOrigin,129.31,81.51,0.00),v40,z0,tPen\WObj:=wPaper;
    MoveL Offs(pOrigin,126.16,84.66,0.00),v40,z0,tPen\WObj:=wPaper;
    MoveL Offs(pOrigin,125.90,84.38,0.00),v40,z0,tPen\WObj:=wPaper;
    MoveL Offs(pOrigin,120.94,79.42,0.00),v40,z0,tPen\WObj:=wPaper;
    MoveL Offs(pOrigin,120.59,79.38,0.00),v40,z0,tPen\WObj:=wPaper;
    MoveL Offs(pOrigin,121.01,79.59,0.00),v40,z0,tPen\WObj:=wPaper;
    MoveL Offs(pOrigin,120.59,79.38,0.00),v40,fine,tPen\WObj:=wPaper;
    MoveL Offs(pOrigin,120.59,79.38,6.00),v60,z5,tPen\WObj:=wPaper;
    MoveL Offs(pOrigin,120.78,78.09,6.00),vTravel,z5,tPen\WObj:=wPaper;
    MoveL Offs(pOrigin,120.78,78.09,0.00),v60,z0,tPen\WObj:=wPaper;
    MoveL Offs(pOrigin,117.03,81.85,0.00),v40,z0,tPen\WObj:=wPaper;
    MoveL Offs(pOrigin,115.98,81.40,0.00),v40,z0,tPen\WObj:=wPaper;
    MoveL Offs(pOrigin,119.89,77.49,0.00),v40,z0,tPen\WObj:=wPaper;
    MoveL Offs(pOrigin,118.99,76.90,0.00),v40,z0,tPen\WObj:=wPaper;
    MoveL Offs(pOrigin,117.49,78.40,0.00),v40,z0,tPen\WObj:=wPaper;
    MoveL Offs(pOrigin,116.74,79.15,0.00),v40,z0,tPen\WObj:=wPaper;
    MoveL Offs(pOrigin,115.08,80.80,0.00),v40,z0,tPen\WObj:=wPaper;
    MoveL Offs(pOrigin,114.04,80.36,0.00),v40,z0,tPen\WObj:=wPaper;
    MoveL Offs(pOrigin,115.84,78.55,0.00),v40,z0,tPen\WObj:=wPaper;
    MoveL Offs(pOrigin,116.59,77.80,0.00),v40,z0,tPen\WObj:=wPaper;
    MoveL Offs(pOrigin,117.94,76.45,0.00),v40,z0,tPen\WObj:=wPaper;
    MoveL Offs(pOrigin,117.05,75.85,0.00),v40,z0,tPen\WObj:=wPaper;
    MoveL Offs(pOrigin,115.99,76.91,0.00),v40,z0,tPen\WObj:=wPaper;
    MoveL Offs(pOrigin,115.10,76.31,0.00),v40,z0,tPen\WObj:=wPaper;
    MoveL Offs(pOrigin,116.30,75.11,0.00),v40,z0,tPen\WObj:=wPaper;
    MoveL Offs(pOrigin,115.40,74.51,0.00),v40,z0,tPen\WObj:=wPaper;
    MoveL Offs(pOrigin,114.50,75.41,0.00),v40,fine,tPen\WObj:=wPaper;
    MoveL Offs(pOrigin,114.50,75.41,6.00),v60,z5,tPen\WObj:=wPaper;
    MoveL Offs(pOrigin,114.94,77.96,6.00),vTravel,z5,tPen\WObj:=wPaper;
    MoveL Offs(pOrigin,114.94,77.96,0.00),v60,z0,tPen\WObj:=wPaper;
    MoveL Offs(pOrigin,113.14,79.76,0.00),v40,fine,tPen\WObj:=wPaper;
    MoveL Offs(pOrigin,113.14,79.76,6.00),v60,z5,tPen\WObj:=wPaper;
    MoveL Offs(pOrigin,112.09,77.04,6.00),vTravel,z5,tPen\WObj:=wPaper;
    MoveL Offs(pOrigin,112.09,77.04,0.00),v60,z0,tPen\WObj:=wPaper;
    MoveL Offs(pOrigin,112.51,77.46,0.00),v40,z0,tPen\WObj:=wPaper;
    MoveL Offs(pOrigin,112.09,77.04,0.00),v40,fine,tPen\WObj:=wPaper;
    MoveL Offs(pOrigin,112.09,77.04,6.00),v60,z5,tPen\WObj:=wPaper;
    MoveL Offs(pOrigin,109.25,79.17,6.00),vTravel,z5,tPen\WObj:=wPaper;
    MoveL Offs(pOrigin,109.25,79.17,0.00),v60,z0,tPen\WObj:=wPaper;
    MoveL Offs(pOrigin,107.59,80.83,0.00),v40,z0,tPen\WObj:=wPaper;
    MoveL Offs(pOrigin,107.00,79.93,0.00),v40,z0,tPen\WObj:=wPaper;
    MoveL Offs(pOrigin,108.35,78.58,0.00),v40,fine,tPen\WObj:=wPaper;
    MoveL Offs(pOrigin,108.35,78.58,6.00),v60,z5,tPen\WObj:=wPaper;
    MoveL Offs(pOrigin,109.96,81.50,6.00),vTravel,z5,tPen\WObj:=wPaper;
    MoveL Offs(pOrigin,109.96,81.50,0.00),v60,z0,tPen\WObj:=wPaper;
    MoveL Offs(pOrigin,110.39,81.93,0.00),v40,z0,tPen\WObj:=wPaper;
    MoveL Offs(pOrigin,109.96,81.50,0.00),v40,fine,tPen\WObj:=wPaper;
    MoveL Offs(pOrigin,109.96,81.50,6.00),v60,z5,tPen\WObj:=wPaper;
    MoveL Offs(pOrigin,108.63,85.77,6.00),vTravel,z5,tPen\WObj:=wPaper;
    MoveL Offs(pOrigin,108.63,85.77,0.00),v60,z0,tPen\WObj:=wPaper;
    MoveL Offs(pOrigin,106.82,87.57,0.00),v40,z0,tPen\WObj:=wPaper;
    MoveL Offs(pOrigin,107.72,88.17,0.00),v40,z0,tPen\WObj:=wPaper;
    MoveL Offs(pOrigin,109.67,86.21,0.00),v40,z0,tPen\WObj:=wPaper;
    MoveL Offs(pOrigin,110.72,86.66,0.00),v40,z0,tPen\WObj:=wPaper;
    MoveL Offs(pOrigin,108.77,88.61,0.00),v40,fine,tPen\WObj:=wPaper;
    MoveL Offs(pOrigin,108.77,88.61,6.00),v60,z5,tPen\WObj:=wPaper;
    MoveL Offs(pOrigin,108.26,86.60,6.00),vTravel,z5,tPen\WObj:=wPaper;
    MoveL Offs(pOrigin,108.26,86.60,0.00),v60,z0,tPen\WObj:=wPaper;
    MoveL Offs(pOrigin,108.69,86.81,0.00),v40,z0,tPen\WObj:=wPaper;
    MoveL Offs(pOrigin,108.26,86.60,0.00),v40,fine,tPen\WObj:=wPaper;
    MoveL Offs(pOrigin,108.26,86.60,6.00),v60,z5,tPen\WObj:=wPaper;
    MoveL Offs(pOrigin,106.35,96.16,6.00),vTravel,z5,tPen\WObj:=wPaper;
    MoveL Offs(pOrigin,106.35,96.16,0.00),v60,z0,tPen\WObj:=wPaper;
    MoveL Offs(pOrigin,106.78,96.38,0.00),v40,z0,tPen\WObj:=wPaper;
    MoveL Offs(pOrigin,106.35,96.16,0.00),v40,fine,tPen\WObj:=wPaper;
    MoveL Offs(pOrigin,106.35,96.16,6.00),v60,z5,tPen\WObj:=wPaper;
    MoveL Offs(pOrigin,109.92,102.39,6.00),vTravel,z5,tPen\WObj:=wPaper;
    MoveL Offs(pOrigin,109.92,102.39,0.00),v60,z0,tPen\WObj:=wPaper;
    MoveL Offs(pOrigin,105.87,106.45,0.00),v40,fine,tPen\WObj:=wPaper;
    MoveL Offs(pOrigin,105.87,106.45,6.00),v60,z5,tPen\WObj:=wPaper;
    MoveL Offs(pOrigin,126.52,89.47,6.00),vTravel,z5,tPen\WObj:=wPaper;
    MoveL Offs(pOrigin,126.52,89.47,0.00),v60,z0,tPen\WObj:=wPaper;
    MoveL Offs(pOrigin,129.52,92.48,0.00),v40,fine,tPen\WObj:=wPaper;
    MoveL Offs(pOrigin,129.52,92.48,6.00),v60,z5,tPen\WObj:=wPaper;
    MoveL Offs(pOrigin,132.58,91.68,6.00),vTravel,z5,tPen\WObj:=wPaper;
    MoveL Offs(pOrigin,132.58,91.68,0.00),v60,z0,tPen\WObj:=wPaper;
    MoveL Offs(pOrigin,144.30,79.96,0.00),v40,fine,tPen\WObj:=wPaper;
    MoveL Offs(pOrigin,144.30,79.96,6.00),v60,z5,tPen\WObj:=wPaper;
    MoveL Offs(pOrigin,145.66,80.24,6.00),vTravel,z5,tPen\WObj:=wPaper;
    MoveL Offs(pOrigin,145.66,80.24,0.00),v60,z0,tPen\WObj:=wPaper;
    MoveL Offs(pOrigin,147.61,82.20,0.00),v40,z0,tPen\WObj:=wPaper;
    MoveL Offs(pOrigin,146.80,81.71,0.00),v40,z0,tPen\WObj:=wPaper;
    MoveL Offs(pOrigin,146.80,80.65,0.00),v40,fine,tPen\WObj:=wPaper;
    MoveL Offs(pOrigin,146.80,80.65,6.00),v60,z5,tPen\WObj:=wPaper;
    MoveL Offs(pOrigin,140.46,84.26,6.00),vTravel,z5,tPen\WObj:=wPaper;
    MoveL Offs(pOrigin,140.46,84.26,0.00),v60,z0,tPen\WObj:=wPaper;
    MoveL Offs(pOrigin,140.46,85.96,0.00),v40,fine,tPen\WObj:=wPaper;
  ENDPROC

